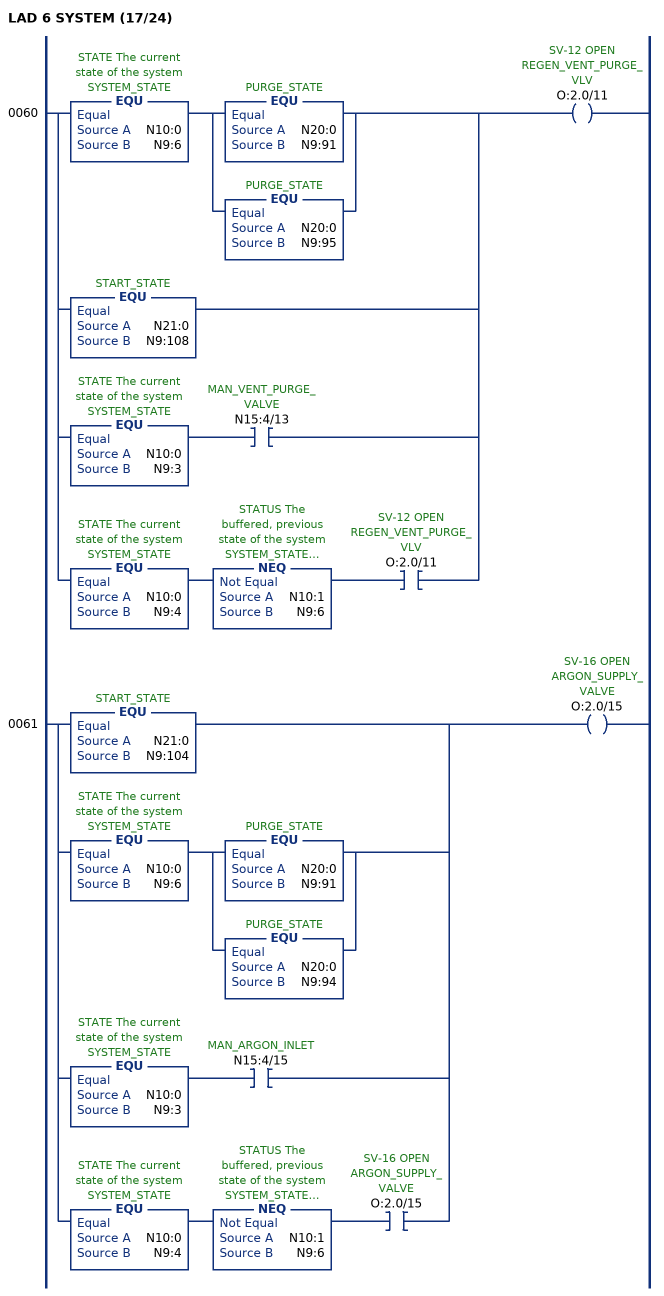
% Rung: 60 %
SOR BST EQU N10:0 N9:6 BST EQU N20:0 N9:91 NXB EQU N20:0 N9:95 BND NXB EQU N21:0 N9:108 NXB EQU N10:0 N9:3 XIC N15:4/13 NXB EQU N10:0 N9:4 NEQ N10:1 N9:6 XIC O:2.0/11 BND OTE O:2.0/11 EOR
%   N10:0  SYSTEM_STATE  "STATE The current state of the system" %
%   N9:6  SYSTEM_PURGE %
%   N20:0  PURGE_STATE %
%   N9:91  PURGE_INIT_VENT %
%   N9:95  PURGE_FINAL_VENT %
%   N21:0  START_STATE %
%   N9:108  START_VENT_GET_2 %
%   N9:3  SYSTEM_MANUAL  "STATE System Manual" %
%   N15:4/13  MAN_VENT_PURGE_VALVE %
%   N9:4  SYSTEM_ALARM  "STATE System Alarm" %
%   N10:1  SYSTEM_STATE_BUFFER  "STATUS The buffered, previous state of the system" %
%   O:2.0/11  REGEN_VENT_PURGE_VLV  "SV-12 OPEN" %
% Rung: 61 %
SOR BST EQU N21:0 N9:104 NXB EQU N10:0 N9:6 BST EQU N20:0 N9:91 NXB EQU N20:0 N9:94 BND NXB EQU N10:0 N9:3 XIC N15:4/15 NXB EQU N10:0 N9:4 NEQ N10:1 N9:6 XIC O:2.0/15 BND OTE O:2.0/15 EOR
%   N21:0  START_STATE %
%   N9:104  START_HEAT %
%   N10:0  SYSTEM_STATE  "STATE The current state of the system" %
%   N9:6  SYSTEM_PURGE %
%   N20:0  PURGE_STATE %
%   N9:91  PURGE_INIT_VENT %
%   N9:94  PURGE_BACKFILL %
%   N9:3  SYSTEM_MANUAL  "STATE System Manual" %
%   N15:4/15  MAN_ARGON_INLET %
%   N9:4  SYSTEM_ALARM  "STATE System Alarm" %
%   N10:1  SYSTEM_STATE_BUFFER  "STATUS The buffered, previous state of the system" %
%   O:2.0/15  ARGON_SUPPLY_VALVE  "SV-16 OPEN" %

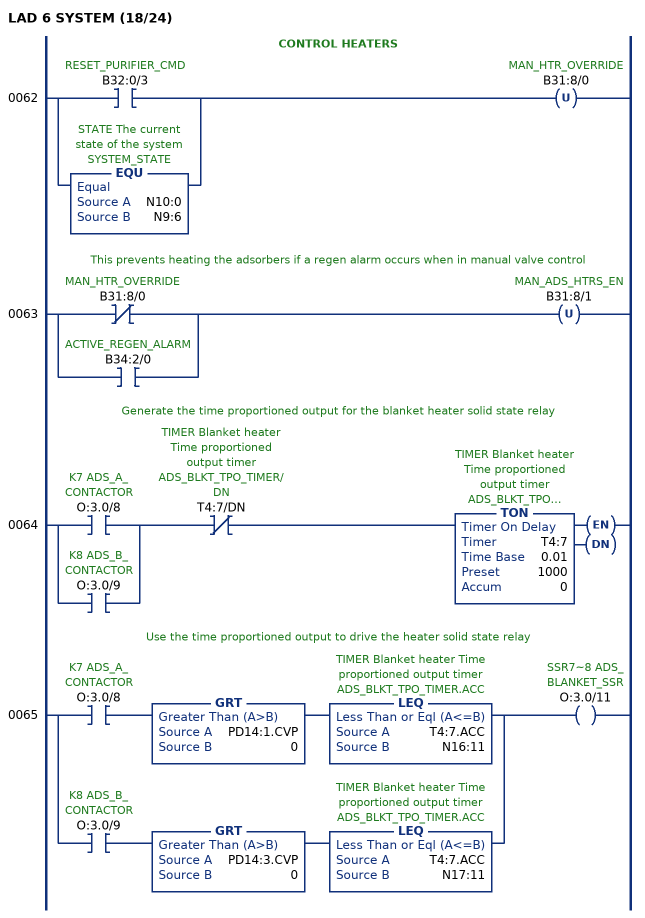
% Rung: 62 %
% TITLE: CONTROL HEATERS %
SOR BST XIC B32:0/3 NXB EQU N10:0 N9:6 BND OTU B31:8/0 EOR
%   B32:0/3  RESET_PURIFIER_CMD %
%   N10:0  SYSTEM_STATE  "STATE The current state of the system" %
%   N9:6  SYSTEM_PURGE %
%   B31:8/0  MAN_HTR_OVERRIDE %
% Rung: 63 %
% This prevents heating the adsorbers if a regen alarm occurs when in manual valve control %
SOR BST XIO B31:8/0 NXB XIC B34:2/0 BND OTU B31:8/1 EOR
%   B31:8/0  MAN_HTR_OVERRIDE %
%   B34:2/0  ACTIVE_REGEN_ALARM %
%   B31:8/1  MAN_ADS_HTRS_EN %
% Rung: 64 %
% Generate the time proportioned output for the blanket heater solid state relay %
SOR BST XIC O:3.0/8 NXB XIC O:3.0/9 BND XIO T4:7/DN TON T4:7 0.01 1000 0 EOR
%   O:3.0/8  ADS_A_CONTACTOR  "K7" %
%   O:3.0/9  ADS_B_CONTACTOR  "K8" %
%   T4:7  ADS_BLKT_TPO_TIMER  "TIMER Blanket heater Time proportioned output timer" %
% Rung: 65 %
% Use the time proportioned output to drive the heater solid state relay %
SOR BST XIC O:3.0/8 GRT PD14:1.CVP 0 LEQ T4:7.ACC N16:11 NXB XIC O:3.0/9 GRT PD14:3.CVP 0 LEQ T4:7.ACC N17:11 BND OTE O:3.0/11 EOR
%   O:3.0/8  ADS_A_CONTACTOR  "K7" %
%   T4:7  ADS_BLKT_TPO_TIMER  "TIMER Blanket heater Time proportioned output timer" %
%   N16:11  ADS_A_BLNKT_OUTPUT  "<datalog> CONTROL ADS A Blanket output (percent)" %
%   O:3.0/9  ADS_B_CONTACTOR  "K8" %
%   N17:11  ADS_B_BLNKT_OUTPUT  "<datalog> CONTROL ADS A Blanket output" %
%   O:3.0/11  ADS_BLANKET_SSR  "SSR7~8" %

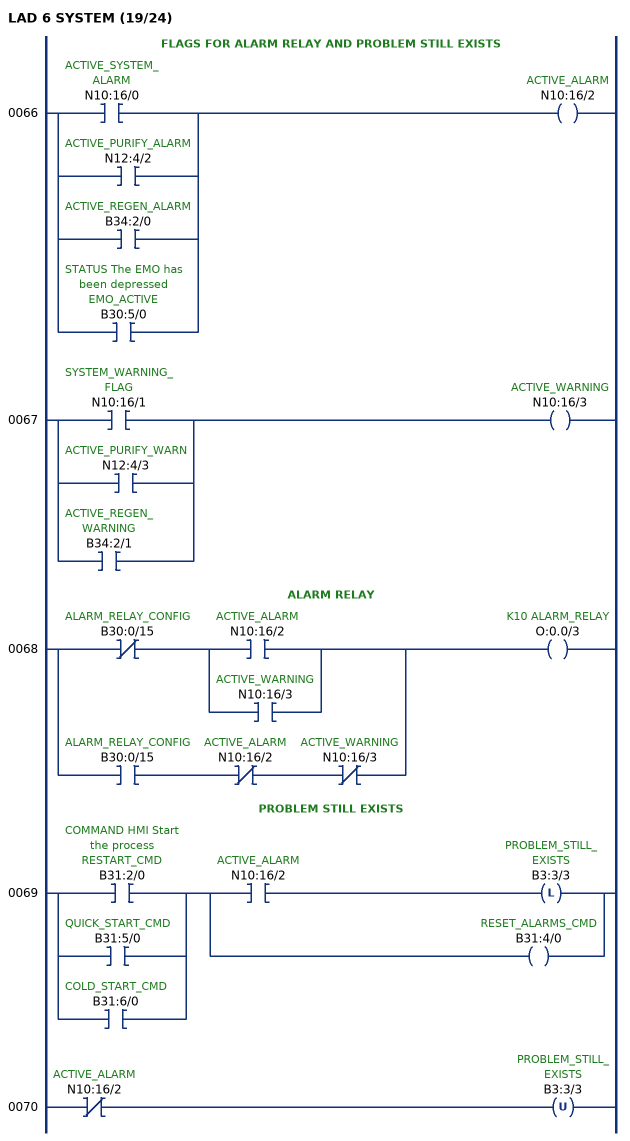
% Rung: 66 %
% TITLE: FLAGS FOR ALARM RELAY AND PROBLEM STILL EXISTS %
SOR BST XIC N10:16/0 NXB XIC N12:4/2 NXB XIC B34:2/0 NXB XIC B30:5/0 BND OTE N10:16/2 EOR
%   N10:16/0  ACTIVE_SYSTEM_ALARM %
%   N12:4/2  ACTIVE_PURIFY_ALARM %
%   B34:2/0  ACTIVE_REGEN_ALARM %
%   B30:5/0  EMO_ACTIVE  "STATUS The EMO has been depressed" %
%   N10:16/2  ACTIVE_ALARM %
% Rung: 67 %
SOR BST XIC N10:16/1 NXB XIC N12:4/3 NXB XIC B34:2/1 BND OTE N10:16/3 EOR
%   N10:16/1  SYSTEM_WARNING_FLAG %
%   N12:4/3  ACTIVE_PURIFY_WARN %
%   B34:2/1  ACTIVE_REGEN_WARNING %
%   N10:16/3  ACTIVE_WARNING %
% Rung: 68 %
% TITLE: ALARM RELAY %
SOR BST XIO B30:0/15 BST XIC N10:16/2 NXB XIC N10:16/3 BND NXB XIC B30:0/15 XIO N10:16/2 XIO N10:16/3 BND OTE O:0.0/3 EOR
%   B30:0/15  ALARM_RELAY_CONFIG %
%   N10:16/2  ACTIVE_ALARM %
%   N10:16/3  ACTIVE_WARNING %
%   O:0.0/3  ALARM_RELAY  "K10" %
% Rung: 69 %
% TITLE: PROBLEM STILL EXISTS %
SOR BST XIC B31:2/0 NXB XIC B31:5/0 NXB XIC B31:6/0 BND BST XIC N10:16/2 OTL B3:3/3 NXB OTE B31:4/0 BND EOR
%   B31:2/0  RESTART_CMD  "COMMAND HMI Start the process" %
%   B31:5/0  QUICK_START_CMD %
%   B31:6/0  COLD_START_CMD %
%   N10:16/2  ACTIVE_ALARM %
%   B3:3/3  PROBLEM_STILL_EXISTS %
%   B31:4/0  RESET_ALARMS_CMD %
% Rung: 70 %
SOR XIO N10:16/2 OTU B3:3/3 EOR
%   N10:16/2  ACTIVE_ALARM %
%   B3:3/3  PROBLEM_STILL_EXISTS %

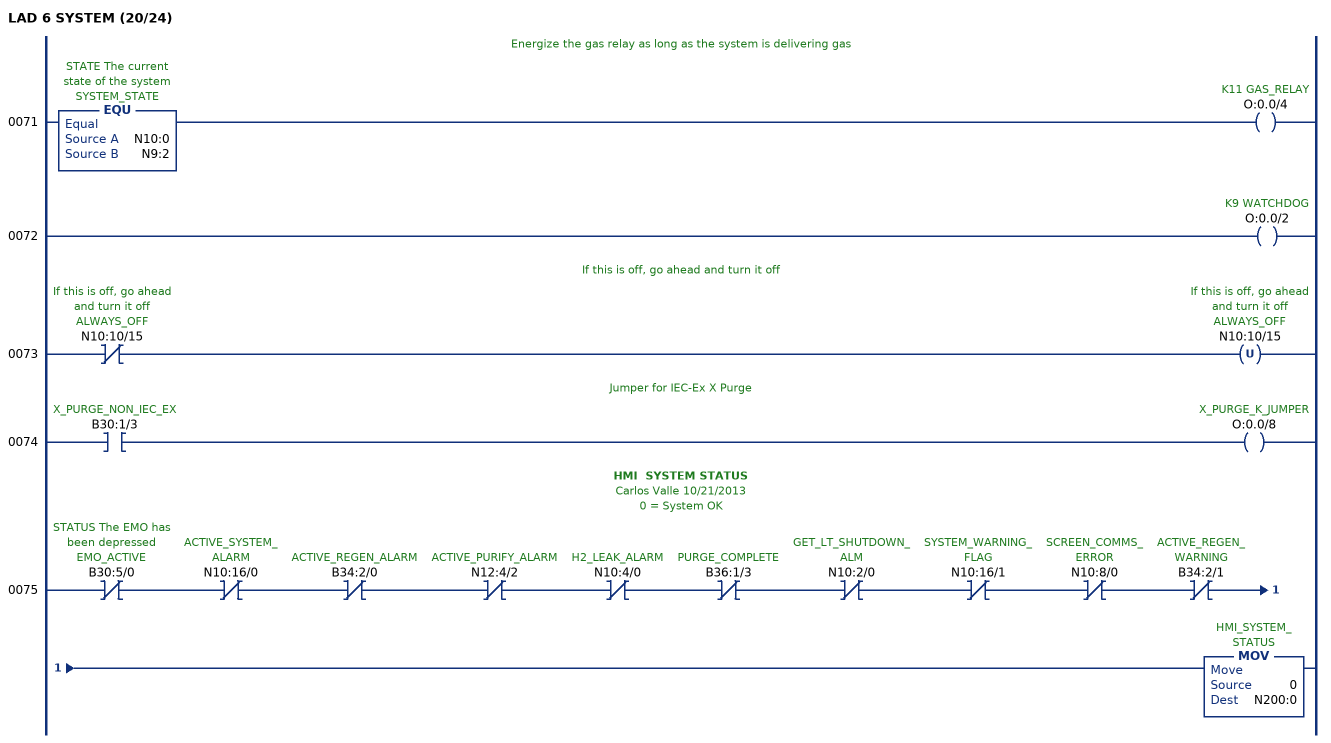
% Rung: 71 %
% Energize the gas relay as long as the system is delivering gas %
SOR EQU N10:0 N9:2 OTE O:0.0/4 EOR
%   N10:0  SYSTEM_STATE  "STATE The current state of the system" %
%   N9:2  SYSTEM_PROCESS  "STATE System Process" %
%   O:0.0/4  GAS_RELAY  "K11" %
% Rung: 72 %
SOR OTE O:0.0/2 EOR
%   O:0.0/2  WATCHDOG  "K9" %
% Rung: 73 %
% If this is off, go ahead and turn it off %
SOR XIO N10:10/15 OTU N10:10/15 EOR
%   N10:10/15  ALWAYS_OFF  "If this is off, go ahead and turn it off" %
% Rung: 74 %
% Jumper for IEC-Ex X Purge %
SOR XIC B30:1/3 OTE O:0.0/8 EOR
%   B30:1/3  X_PURGE_NON_IEC_EX %
%   O:0.0/8  X_PURGE_K_JUMPER %
% Rung: 75 %
% TITLE: HMI  SYSTEM STATUS %
% Carlos Valle 10/21/2013
% 0 = System OK %
SOR XIO B30:5/0 XIO N10:16/0 XIO B34:2/0 XIO N12:4/2 XIO N10:4/0 XIO B36:1/3 XIO N10:2/0 XIO N10:16/1 XIO N10:8/0 XIO B34:2/1 MOV 0 N200:0 EOR
%   B30:5/0  EMO_ACTIVE  "STATUS The EMO has been depressed" %
%   N10:16/0  ACTIVE_SYSTEM_ALARM %
%   B34:2/0  ACTIVE_REGEN_ALARM %
%   N12:4/2  ACTIVE_PURIFY_ALARM %
%   N10:4/0  H2_LEAK_ALARM %
%   B36:1/3  PURGE_COMPLETE %
%   N10:2/0  GET_LT_SHUTDOWN_ALM %
%   N10:16/1  SYSTEM_WARNING_FLAG %
%   N10:8/0  SCREEN_COMMS_ERROR %
%   B34:2/1  ACTIVE_REGEN_WARNING %
%   N200:0  HMI_SYSTEM_STATUS %

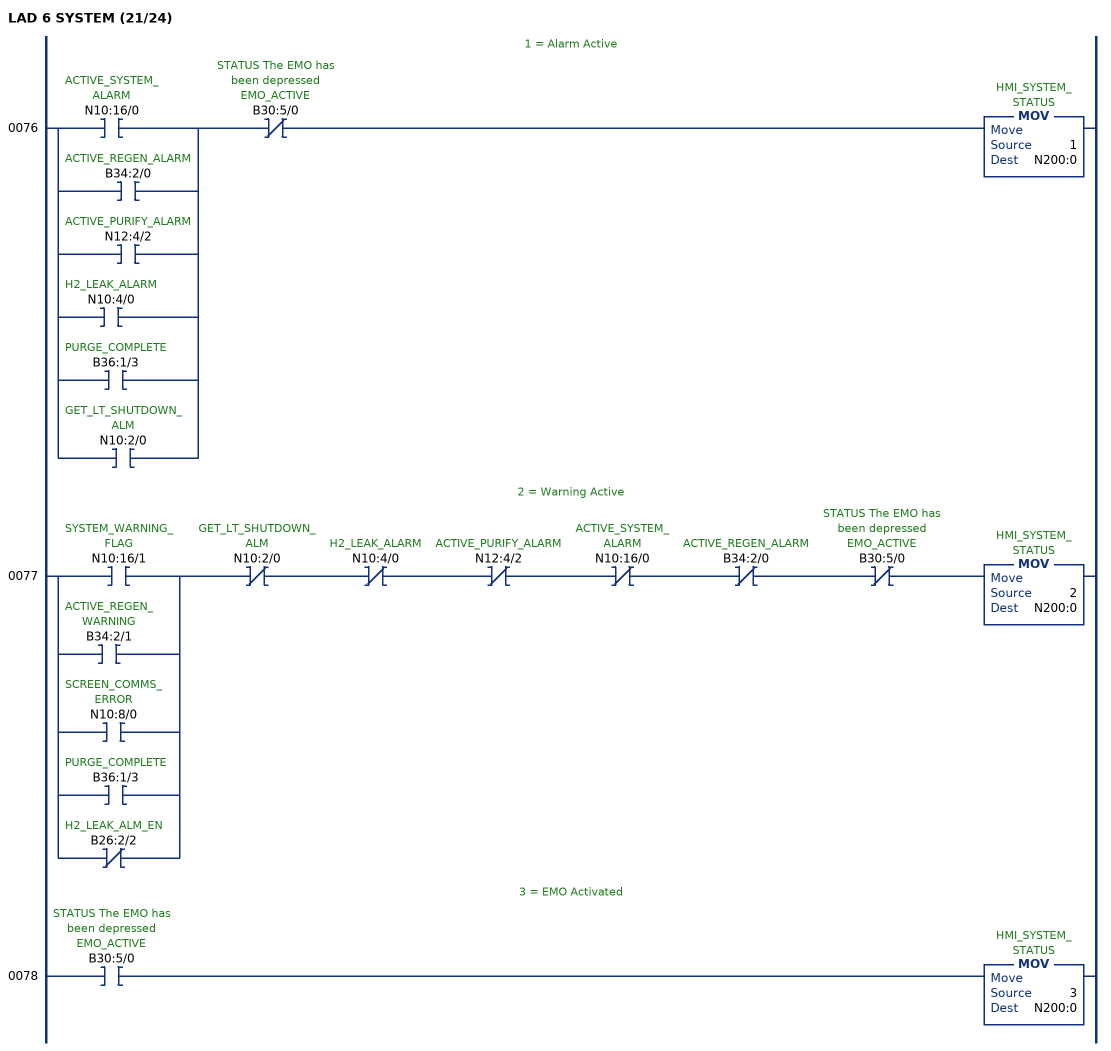
% Rung: 76 %
% 1 = Alarm Active %
SOR BST XIC N10:16/0 NXB XIC B34:2/0 NXB XIC N12:4/2 NXB XIC N10:4/0 NXB XIC B36:1/3 NXB XIC N10:2/0 BND XIO B30:5/0 MOV 1 N200:0 EOR
%   N10:16/0  ACTIVE_SYSTEM_ALARM %
%   B34:2/0  ACTIVE_REGEN_ALARM %
%   N12:4/2  ACTIVE_PURIFY_ALARM %
%   N10:4/0  H2_LEAK_ALARM %
%   B36:1/3  PURGE_COMPLETE %
%   N10:2/0  GET_LT_SHUTDOWN_ALM %
%   B30:5/0  EMO_ACTIVE  "STATUS The EMO has been depressed" %
%   N200:0  HMI_SYSTEM_STATUS %
% Rung: 77 %
% 2 = Warning Active %
SOR BST XIC N10:16/1 NXB XIC B34:2/1 NXB XIC N10:8/0 NXB XIC B36:1/3 NXB XIO B26:2/2 BND XIO N10:2/0 XIO N10:4/0 XIO N12:4/2 XIO N10:16/0 XIO B34:2/0 XIO B30:5/0 MOV 2 N200:0 EOR
%   N10:16/1  SYSTEM_WARNING_FLAG %
%   B34:2/1  ACTIVE_REGEN_WARNING %
%   N10:8/0  SCREEN_COMMS_ERROR %
%   B36:1/3  PURGE_COMPLETE %
%   B26:2/2  H2_LEAK_ALM_EN %
%   N10:2/0  GET_LT_SHUTDOWN_ALM %
%   N10:4/0  H2_LEAK_ALARM %
%   N12:4/2  ACTIVE_PURIFY_ALARM %
%   N10:16/0  ACTIVE_SYSTEM_ALARM %
%   B34:2/0  ACTIVE_REGEN_ALARM %
%   B30:5/0  EMO_ACTIVE  "STATUS The EMO has been depressed" %
%   N200:0  HMI_SYSTEM_STATUS %
% Rung: 78 %
% 3 = EMO Activated %
SOR XIC B30:5/0 MOV 3 N200:0 EOR
%   B30:5/0  EMO_ACTIVE  "STATUS The EMO has been depressed" %
%   N200:0  HMI_SYSTEM_STATUS %

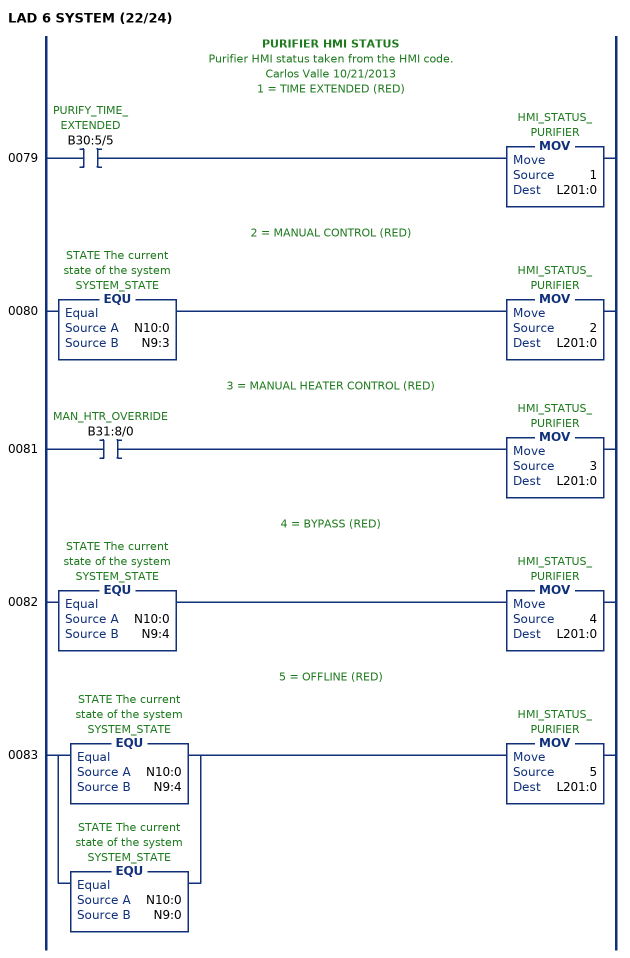
% Rung: 79 %
% TITLE: PURIFIER HMI STATUS %
% Purifier HMI status taken from the HMI code.
% Carlos Valle 10/21/2013
% 1 = TIME EXTENDED (RED) %
SOR XIC B30:5/5 MOV 1 L201:0 EOR
%   B30:5/5  PURIFY_TIME_EXTENDED %
%   L201:0  HMI_STATUS_PURIFIER %
% Rung: 80 %
% 2 = MANUAL CONTROL (RED) %
SOR EQU N10:0 N9:3 MOV 2 L201:0 EOR
%   N10:0  SYSTEM_STATE  "STATE The current state of the system" %
%   N9:3  SYSTEM_MANUAL  "STATE System Manual" %
%   L201:0  HMI_STATUS_PURIFIER %
% Rung: 81 %
% 3 = MANUAL HEATER CONTROL (RED) %
SOR XIC B31:8/0 MOV 3 L201:0 EOR
%   B31:8/0  MAN_HTR_OVERRIDE %
%   L201:0  HMI_STATUS_PURIFIER %
% Rung: 82 %
% 4 = BYPASS (RED) %
SOR EQU N10:0 N9:4 MOV 4 L201:0 EOR
%   N10:0  SYSTEM_STATE  "STATE The current state of the system" %
%   N9:4  SYSTEM_ALARM  "STATE System Alarm" %
%   L201:0  HMI_STATUS_PURIFIER %
% Rung: 83 %
% 5 = OFFLINE (RED) %
SOR BST EQU N10:0 N9:4 NXB EQU N10:0 N9:0 BND MOV 5 L201:0 EOR
%   N10:0  SYSTEM_STATE  "STATE The current state of the system" %
%   N9:4  SYSTEM_ALARM  "STATE System Alarm" %
%   N9:0  SYSTEM_OFFLINE %
%   L201:0  HMI_STATUS_PURIFIER %

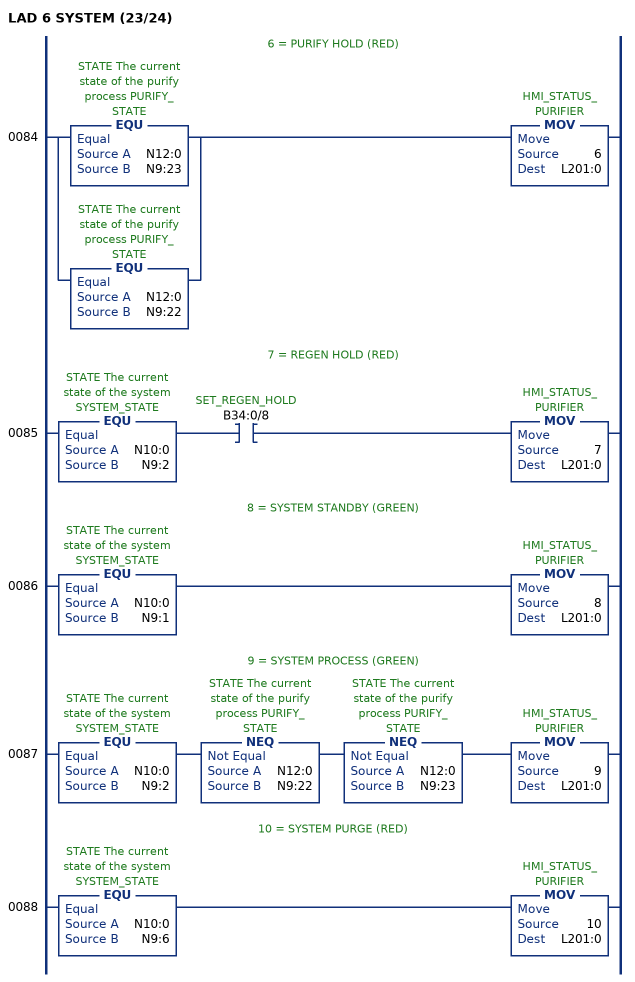
% Rung: 84 %
% 6 = PURIFY HOLD (RED) %
SOR BST EQU N12:0 N9:23 NXB EQU N12:0 N9:22 BND MOV 6 L201:0 EOR
%   N12:0  PURIFY_STATE  "STATE The current state of the purify process" %
%   N9:23  PURIFY_MANUAL_HOLD  "STATE Purify Manual Hold" %
%   N9:22  PURIFY_HOLD  "STATE Purify Hold" %
%   L201:0  HMI_STATUS_PURIFIER %
% Rung: 85 %
% 7 = REGEN HOLD (RED) %
SOR EQU N10:0 N9:2 XIC B34:0/8 MOV 7 L201:0 EOR
%   N10:0  SYSTEM_STATE  "STATE The current state of the system" %
%   N9:2  SYSTEM_PROCESS  "STATE System Process" %
%   B34:0/8  SET_REGEN_HOLD %
%   L201:0  HMI_STATUS_PURIFIER %
% Rung: 86 %
% 8 = SYSTEM STANDBY (GREEN) %
SOR EQU N10:0 N9:1 MOV 8 L201:0 EOR
%   N10:0  SYSTEM_STATE  "STATE The current state of the system" %
%   N9:1  SYSTEM_STANDBY  "STATE System Process" %
%   L201:0  HMI_STATUS_PURIFIER %
% Rung: 87 %
% 9 = SYSTEM PROCESS (GREEN) %
SOR EQU N10:0 N9:2 NEQ N12:0 N9:22 NEQ N12:0 N9:23 MOV 9 L201:0 EOR
%   N10:0  SYSTEM_STATE  "STATE The current state of the system" %
%   N9:2  SYSTEM_PROCESS  "STATE System Process" %
%   N12:0  PURIFY_STATE  "STATE The current state of the purify process" %
%   N9:22  PURIFY_HOLD  "STATE Purify Hold" %
%   N9:23  PURIFY_MANUAL_HOLD  "STATE Purify Manual Hold" %
%   L201:0  HMI_STATUS_PURIFIER %
% Rung: 88 %
% 10 = SYSTEM PURGE (RED) %
SOR EQU N10:0 N9:6 MOV 10 L201:0 EOR
%   N10:0  SYSTEM_STATE  "STATE The current state of the system" %
%   N9:6  SYSTEM_PURGE %
%   L201:0  HMI_STATUS_PURIFIER %

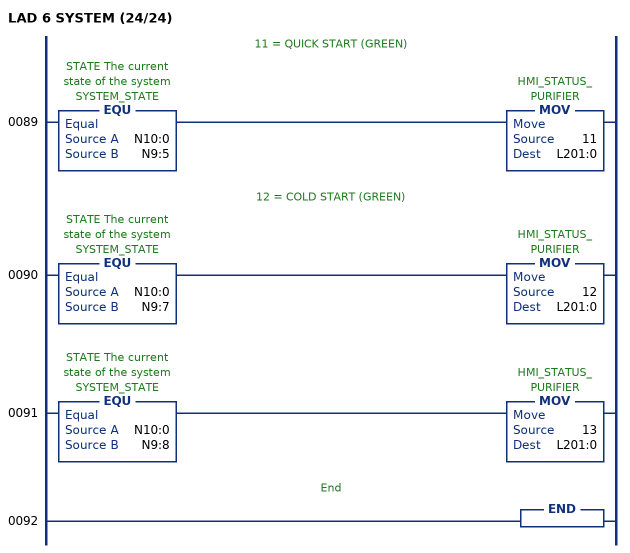
% Rung: 89 %
% 11 = QUICK START (GREEN) %
SOR EQU N10:0 N9:5 MOV 11 L201:0 EOR
%   N10:0  SYSTEM_STATE  "STATE The current state of the system" %
%   N9:5  SYSTEM_QUICK_START %
%   L201:0  HMI_STATUS_PURIFIER %
% Rung: 90 %
% 12 = COLD START (GREEN) %
SOR EQU N10:0 N9:7 MOV 12 L201:0 EOR
%   N10:0  SYSTEM_STATE  "STATE The current state of the system" %
%   N9:7  SYSTEM_COLD_START %
%   L201:0  HMI_STATUS_PURIFIER %
% Rung: 91 %
SOR EQU N10:0 N9:8 MOV 13 L201:0 EOR
%   N10:0  SYSTEM_STATE  "STATE The current state of the system" %
%   N9:8  SYSTEM_SUPPLEMENTAL %
%   L201:0  HMI_STATUS_PURIFIER %
% Rung: 92 %
% End %
SOR END EOR

LADDER 7 "PROCESSING"    % Runs the processing control %
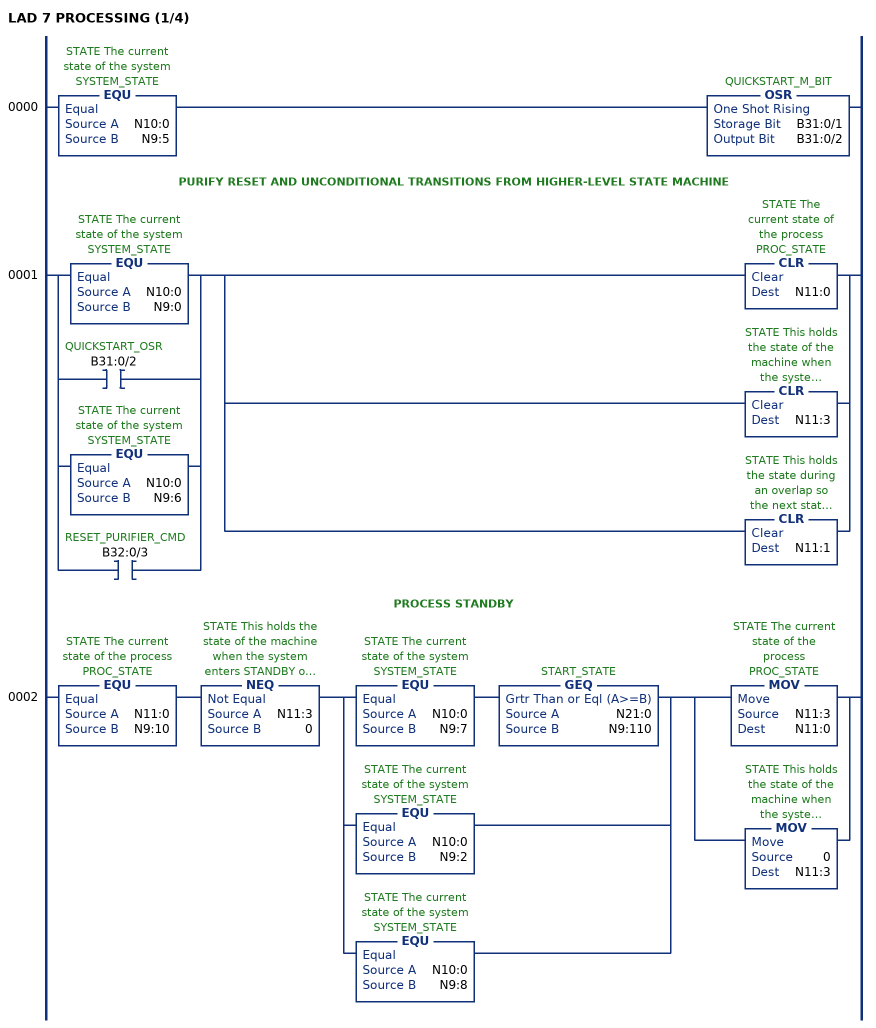
% Rung: 0 %
SOR EQU N10:0 N9:5 OSR B31:0/1 B31:0/2 EOR
%   N10:0  SYSTEM_STATE  "STATE The current state of the system" %
%   N9:5  SYSTEM_QUICK_START %
%   B31:0/1  QUICKSTART_M_BIT %
%   B31:0/2  QUICKSTART_OSR %
% Rung: 1 %
% TITLE: PURIFY RESET AND UNCONDITIONAL TRANSITIONS FROM HIGHER-LEVEL STATE MACHINE %
SOR BST EQU N10:0 N9:0 NXB XIC B31:0/2 NXB EQU N10:0 N9:6 NXB XIC B32:0/3 BND BST CLR N11:0 NXB CLR N11:3 NXB CLR N11:1 BND EOR
%   N10:0  SYSTEM_STATE  "STATE The current state of the system" %
%   N9:0  SYSTEM_OFFLINE %
%   B31:0/2  QUICKSTART_OSR %
%   N9:6  SYSTEM_PURGE %
%   B32:0/3  RESET_PURIFIER_CMD %
%   N11:0  PROC_STATE  "STATE The current state of the process" %
%   N11:3  PROC_STATE_BUFFER  "STATE This holds the state of the machine when the system enters STANDBY or ALARM" %
%   N11:1  PROC_OVERLAP_BUFFER  "STATE This holds the state during an overlap so the next state can be determined" %
% Rung: 2 %
% TITLE: PROCESS STANDBY %
SOR EQU N11:0 N9:10 NEQ N11:3 0 BST EQU N10:0 N9:7 GEQ N21:0 N9:110 NXB EQU N10:0 N9:2 NXB EQU N10:0 N9:8 BND BST MOV N11:3 N11:0 NXB MOV 0 N11:3 BND EOR
%   N11:0  PROC_STATE  "STATE The current state of the process" %
%   N9:10  PROC_STANDBY  "STATE Process Standby" %
%   N11:3  PROC_STATE_BUFFER  "STATE This holds the state of the machine when the system enters STANDBY or ALARM" %
%   N10:0  SYSTEM_STATE  "STATE The current state of the system" %
%   N9:7  SYSTEM_COLD_START %
%   N21:0  START_STATE %
%   N9:110  START_REG_VENT %
%   N9:2  SYSTEM_PROCESS  "STATE System Process" %
%   N9:8  SYSTEM_SUPPLEMENTAL %

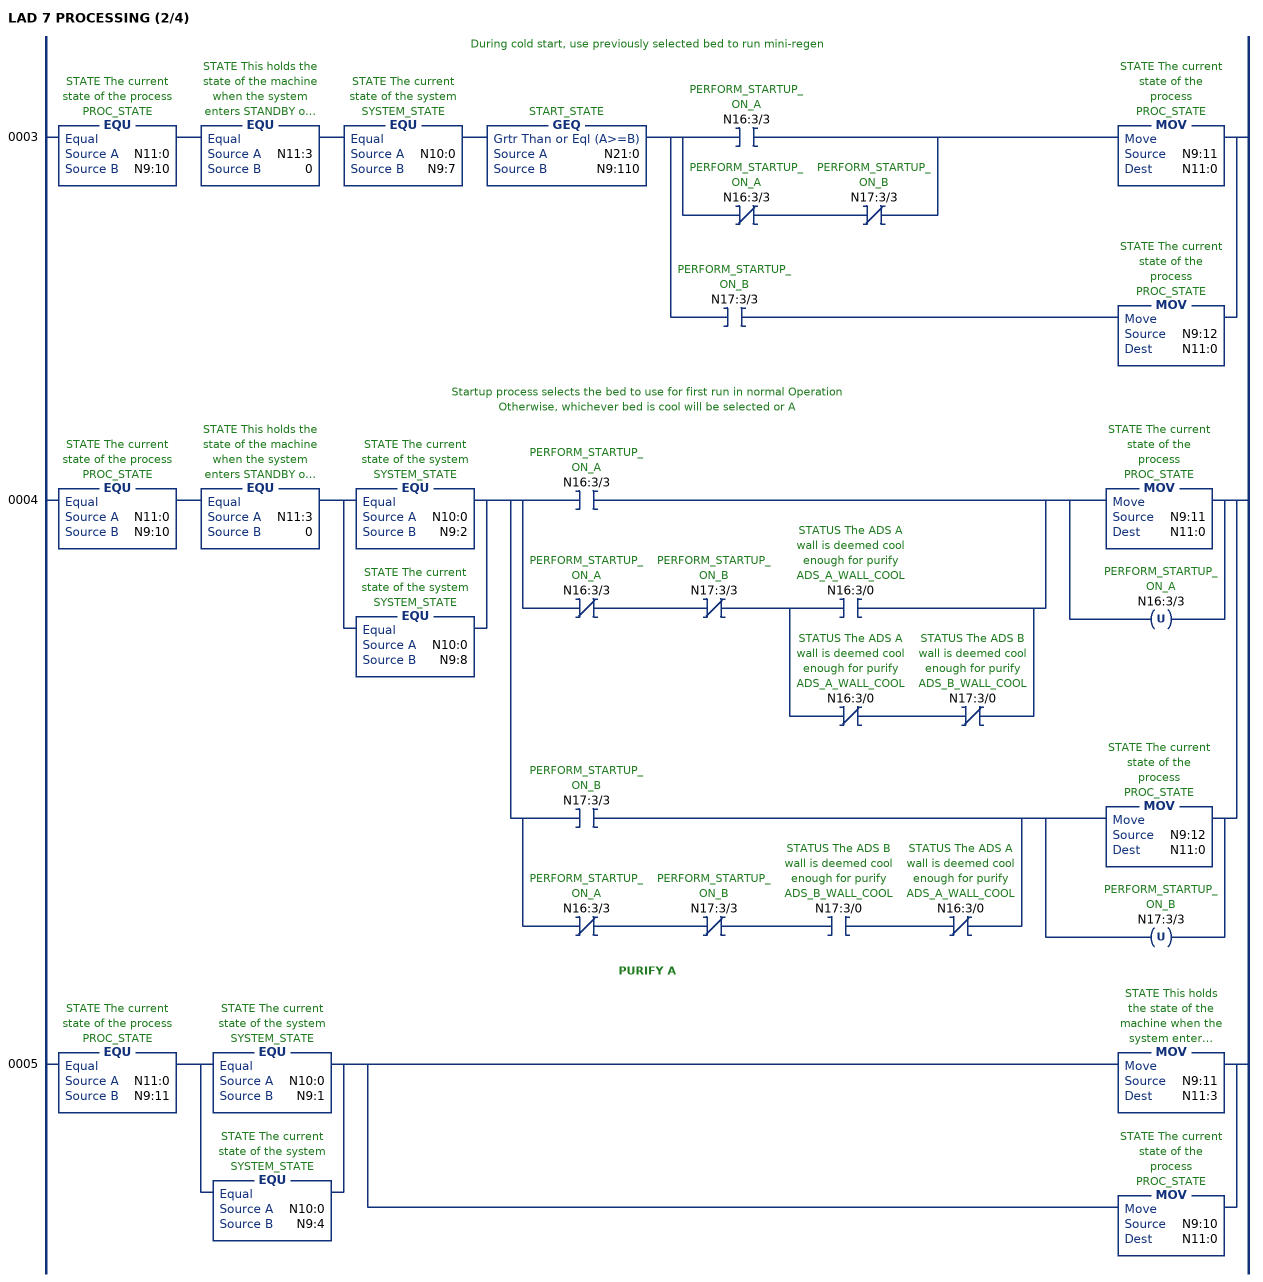
% Rung: 3 %
% During cold start, use previously selected bed to run mini-regen %
SOR EQU N11:0 N9:10 EQU N11:3 0 EQU N10:0 N9:7 GEQ N21:0 N9:110 BST BST XIC N16:3/3 NXB XIO N16:3/3 XIO N17:3/3 BND MOV N9:11 N11:0 NXB XIC N17:3/3 MOV N9:12 N11:0 BND EOR
%   N11:0  PROC_STATE  "STATE The current state of the process" %
%   N9:10  PROC_STANDBY  "STATE Process Standby" %
%   N11:3  PROC_STATE_BUFFER  "STATE This holds the state of the machine when the system enters STANDBY or ALARM" %
%   N10:0  SYSTEM_STATE  "STATE The current state of the system" %
%   N9:7  SYSTEM_COLD_START %
%   N21:0  START_STATE %
%   N9:110  START_REG_VENT %
%   N16:3/3  PERFORM_STARTUP_ON_A %
%   N17:3/3  PERFORM_STARTUP_ON_B %
%   N9:11  PROC_PFY_A_REG_B  "STATE Process Purify A" %
%   N9:12  PROC_PFY_B_REG_A  "STATE Process Purify B" %
% Rung: 4 %
% Startup process selects the bed to use for first run in normal Operation
% Otherwise, whichever bed is cool will be selected or A %
SOR EQU N11:0 N9:10 EQU N11:3 0 BST EQU N10:0 N9:2 NXB EQU N10:0 N9:8 BND BST BST XIC N16:3/3 NXB XIO N16:3/3 XIO N17:3/3 BST XIC N16:3/0 NXB XIO N16:3/0 XIO N17:3/0 BND BND BST MOV N9:11 N11:0 NXB OTU N16:3/3 BND NXB BST XIC N17:3/3 NXB XIO N16:3/3 XIO N17:3/3 XIC N17:3/0 XIO N16:3/0 BND BST MOV N9:12 N11:0 NXB OTU N17:3/3 BND BND EOR
%   N11:0  PROC_STATE  "STATE The current state of the process" %
%   N9:10  PROC_STANDBY  "STATE Process Standby" %
%   N11:3  PROC_STATE_BUFFER  "STATE This holds the state of the machine when the system enters STANDBY or ALARM" %
%   N10:0  SYSTEM_STATE  "STATE The current state of the system" %
%   N9:2  SYSTEM_PROCESS  "STATE System Process" %
%   N9:8  SYSTEM_SUPPLEMENTAL %
%   N16:3/3  PERFORM_STARTUP_ON_A %
%   N17:3/3  PERFORM_STARTUP_ON_B %
%   N16:3/0  ADS_A_WALL_COOL  "STATUS The ADS A wall is deemed cool enough for purify" %
%   N17:3/0  ADS_B_WALL_COOL  "STATUS The ADS B wall is deemed cool enough for purify" %
%   N9:11  PROC_PFY_A_REG_B  "STATE Process Purify A" %
%   N9:12  PROC_PFY_B_REG_A  "STATE Process Purify B" %
% Rung: 5 %
% TITLE: PURIFY A %
SOR EQU N11:0 N9:11 BST EQU N10:0 N9:1 NXB EQU N10:0 N9:4 BND BST MOV N9:11 N11:3 NXB MOV N9:10 N11:0 BND EOR
%   N11:0  PROC_STATE  "STATE The current state of the process" %
%   N9:11  PROC_PFY_A_REG_B  "STATE Process Purify A" %
%   N10:0  SYSTEM_STATE  "STATE The current state of the system" %
%   N9:1  SYSTEM_STANDBY  "STATE System Process" %
%   N9:4  SYSTEM_ALARM  "STATE System Alarm" %
%   N11:3  PROC_STATE_BUFFER  "STATE This holds the state of the machine when the system enters STANDBY or ALARM" %
%   N9:10  PROC_STANDBY  "STATE Process Standby" %

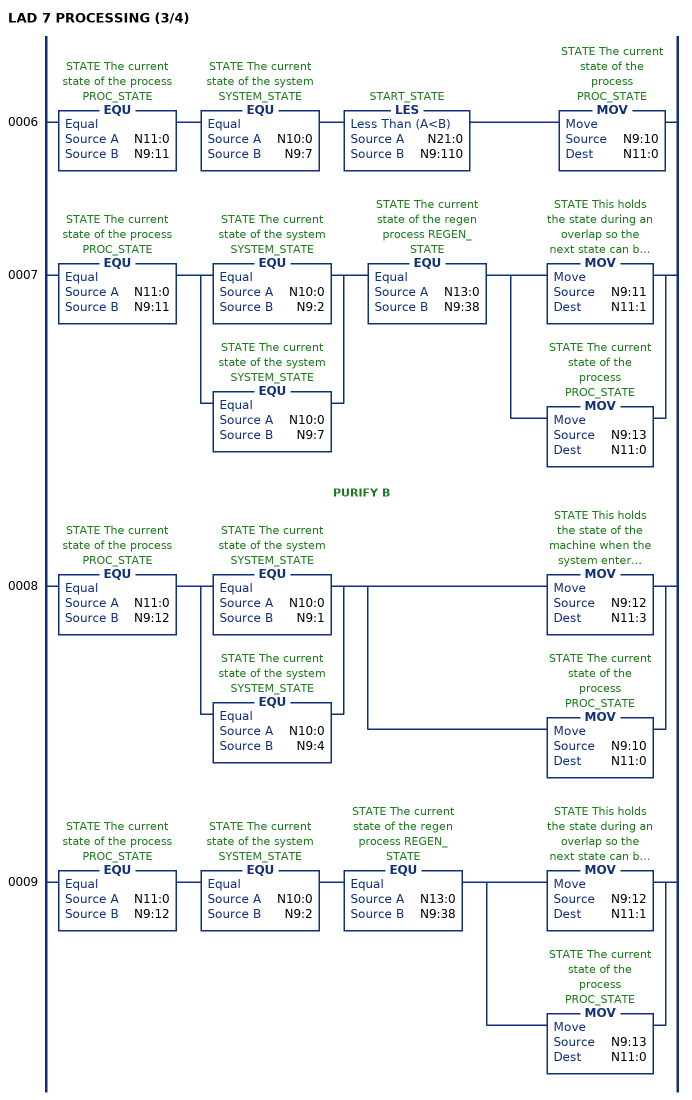
% Rung: 6 %
SOR EQU N11:0 N9:11 EQU N10:0 N9:7 LES N21:0 N9:110 MOV N9:10 N11:0 EOR
%   N11:0  PROC_STATE  "STATE The current state of the process" %
%   N9:11  PROC_PFY_A_REG_B  "STATE Process Purify A" %
%   N10:0  SYSTEM_STATE  "STATE The current state of the system" %
%   N9:7  SYSTEM_COLD_START %
%   N21:0  START_STATE %
%   N9:110  START_REG_VENT %
%   N9:10  PROC_STANDBY  "STATE Process Standby" %
% Rung: 7 %
SOR EQU N11:0 N9:11 BST EQU N10:0 N9:2 NXB EQU N10:0 N9:7 BND EQU N13:0 N9:38 BST MOV N9:11 N11:1 NXB MOV N9:13 N11:0 BND EOR
%   N11:0  PROC_STATE  "STATE The current state of the process" %
%   N9:11  PROC_PFY_A_REG_B  "STATE Process Purify A" %
%   N10:0  SYSTEM_STATE  "STATE The current state of the system" %
%   N9:2  SYSTEM_PROCESS  "STATE System Process" %
%   N9:7  SYSTEM_COLD_START %
%   N13:0  REGEN_STATE  "STATE The current state of the regen process" %
%   N9:38  REGEN_DONE %
%   N11:1  PROC_OVERLAP_BUFFER  "STATE This holds the state during an overlap so the next state can be determined" %
%   N9:13  PROC_OVERLAP  "STATE Process Purify Overlap" %
% Rung: 8 %
% TITLE: PURIFY B %
SOR EQU N11:0 N9:12 BST EQU N10:0 N9:1 NXB EQU N10:0 N9:4 BND BST MOV N9:12 N11:3 NXB MOV N9:10 N11:0 BND EOR
%   N11:0  PROC_STATE  "STATE The current state of the process" %
%   N9:12  PROC_PFY_B_REG_A  "STATE Process Purify B" %
%   N10:0  SYSTEM_STATE  "STATE The current state of the system" %
%   N9:1  SYSTEM_STANDBY  "STATE System Process" %
%   N9:4  SYSTEM_ALARM  "STATE System Alarm" %
%   N11:3  PROC_STATE_BUFFER  "STATE This holds the state of the machine when the system enters STANDBY or ALARM" %
%   N9:10  PROC_STANDBY  "STATE Process Standby" %
% Rung: 9 %
SOR EQU N11:0 N9:12 EQU N10:0 N9:2 EQU N13:0 N9:38 BST MOV N9:12 N11:1 NXB MOV N9:13 N11:0 BND EOR
%   N11:0  PROC_STATE  "STATE The current state of the process" %
%   N9:12  PROC_PFY_B_REG_A  "STATE Process Purify B" %
%   N10:0  SYSTEM_STATE  "STATE The current state of the system" %
%   N9:2  SYSTEM_PROCESS  "STATE System Process" %
%   N13:0  REGEN_STATE  "STATE The current state of the regen process" %
%   N9:38  REGEN_DONE %
%   N11:1  PROC_OVERLAP_BUFFER  "STATE This holds the state during an overlap so the next state can be determined" %
%   N9:13  PROC_OVERLAP  "STATE Process Purify Overlap" %

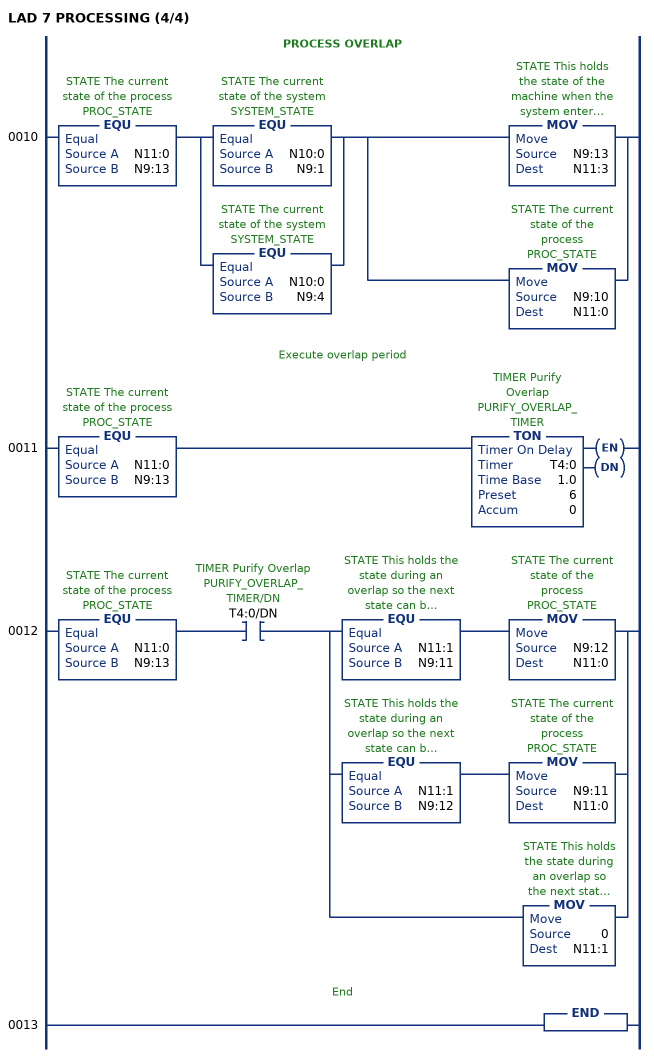
% Rung: 10 %
% TITLE: PROCESS OVERLAP %
SOR EQU N11:0 N9:13 BST EQU N10:0 N9:1 NXB EQU N10:0 N9:4 BND BST MOV N9:13 N11:3 NXB MOV N9:10 N11:0 BND EOR
%   N11:0  PROC_STATE  "STATE The current state of the process" %
%   N9:13  PROC_OVERLAP  "STATE Process Purify Overlap" %
%   N10:0  SYSTEM_STATE  "STATE The current state of the system" %
%   N9:1  SYSTEM_STANDBY  "STATE System Process" %
%   N9:4  SYSTEM_ALARM  "STATE System Alarm" %
%   N11:3  PROC_STATE_BUFFER  "STATE This holds the state of the machine when the system enters STANDBY or ALARM" %
%   N9:10  PROC_STANDBY  "STATE Process Standby" %
% Rung: 11 %
% Execute overlap period %
SOR EQU N11:0 N9:13 TON T4:0 1.0 6 0 EOR
%   N11:0  PROC_STATE  "STATE The current state of the process" %
%   N9:13  PROC_OVERLAP  "STATE Process Purify Overlap" %
%   T4:0  PURIFY_OVERLAP_TIMER  "TIMER Purify Overlap" %
% Rung: 12 %
SOR EQU N11:0 N9:13 XIC T4:0/DN BST EQU N11:1 N9:11 MOV N9:12 N11:0 NXB EQU N11:1 N9:12 MOV N9:11 N11:0 NXB MOV 0 N11:1 BND EOR
%   N11:0  PROC_STATE  "STATE The current state of the process" %
%   N9:13  PROC_OVERLAP  "STATE Process Purify Overlap" %
%   T4:0  PURIFY_OVERLAP_TIMER  "TIMER Purify Overlap" %
%   N11:1  PROC_OVERLAP_BUFFER  "STATE This holds the state during an overlap so the next state can be determined" %
%   N9:11  PROC_PFY_A_REG_B  "STATE Process Purify A" %
%   N9:12  PROC_PFY_B_REG_A  "STATE Process Purify B" %
% Rung: 13 %
% End %
SOR END EOR

LADDER 8 "MANUAL_CTL"    % Runs the manual valve control %
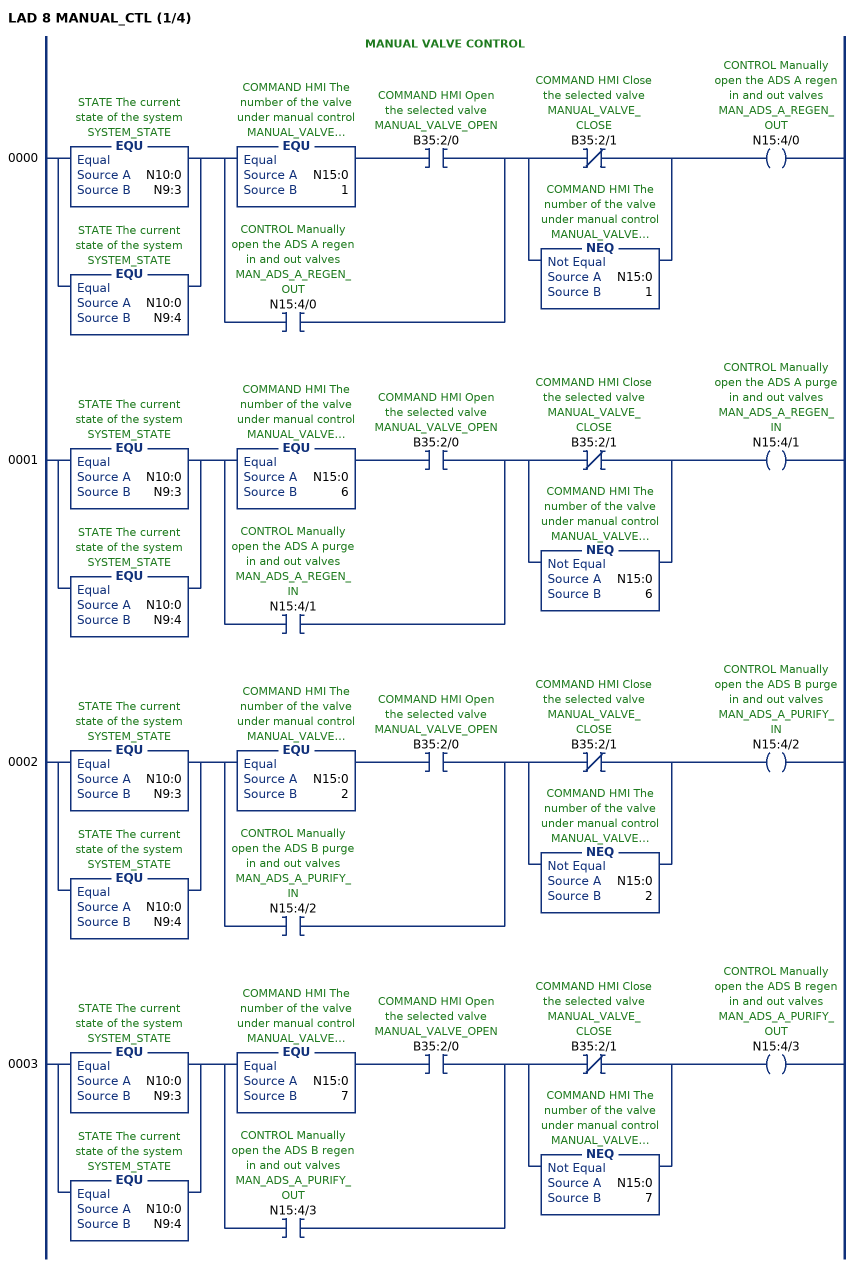
% Rung: 0 %
% TITLE: MANUAL VALVE CONTROL %
SOR BST EQU N10:0 N9:3 NXB EQU N10:0 N9:4 BND BST EQU N15:0 1 XIC B35:2/0 NXB XIC N15:4/0 BND BST XIO B35:2/1 NXB NEQ N15:0 1 BND OTE N15:4/0 EOR
%   N10:0  SYSTEM_STATE  "STATE The current state of the system" %
%   N9:3  SYSTEM_MANUAL  "STATE System Manual" %
%   N9:4  SYSTEM_ALARM  "STATE System Alarm" %
%   N15:0  MANUAL_VALVE_NUMBER  "COMMAND HMI The number of the valve under manual control" %
%   B35:2/0  MANUAL_VALVE_OPEN  "COMMAND HMI Open the selected valve" %
%   N15:4/0  MAN_ADS_A_REGEN_OUT  "CONTROL Manually open the ADS A regen in and out valves" %
%   B35:2/1  MANUAL_VALVE_CLOSE  "COMMAND HMI Close the selected valve" %
% Rung: 1 %
SOR BST EQU N10:0 N9:3 NXB EQU N10:0 N9:4 BND BST EQU N15:0 6 XIC B35:2/0 NXB XIC N15:4/1 BND BST XIO B35:2/1 NXB NEQ N15:0 6 BND OTE N15:4/1 EOR
%   N10:0  SYSTEM_STATE  "STATE The current state of the system" %
%   N9:3  SYSTEM_MANUAL  "STATE System Manual" %
%   N9:4  SYSTEM_ALARM  "STATE System Alarm" %
%   N15:0  MANUAL_VALVE_NUMBER  "COMMAND HMI The number of the valve under manual control" %
%   B35:2/0  MANUAL_VALVE_OPEN  "COMMAND HMI Open the selected valve" %
%   N15:4/1  MAN_ADS_A_REGEN_IN  "CONTROL Manually open the ADS A purge in and out valves" %
%   B35:2/1  MANUAL_VALVE_CLOSE  "COMMAND HMI Close the selected valve" %
% Rung: 2 %
SOR BST EQU N10:0 N9:3 NXB EQU N10:0 N9:4 BND BST EQU N15:0 2 XIC B35:2/0 NXB XIC N15:4/2 BND BST XIO B35:2/1 NXB NEQ N15:0 2 BND OTE N15:4/2 EOR
%   N10:0  SYSTEM_STATE  "STATE The current state of the system" %
%   N9:3  SYSTEM_MANUAL  "STATE System Manual" %
%   N9:4  SYSTEM_ALARM  "STATE System Alarm" %
%   N15:0  MANUAL_VALVE_NUMBER  "COMMAND HMI The number of the valve under manual control" %
%   B35:2/0  MANUAL_VALVE_OPEN  "COMMAND HMI Open the selected valve" %
%   N15:4/2  MAN_ADS_A_PURIFY_IN  "CONTROL Manually open the ADS B purge in and out valves" %
%   B35:2/1  MANUAL_VALVE_CLOSE  "COMMAND HMI Close the selected valve" %
% Rung: 3 %
SOR BST EQU N10:0 N9:3 NXB EQU N10:0 N9:4 BND BST EQU N15:0 7 XIC B35:2/0 NXB XIC N15:4/3 BND BST XIO B35:2/1 NXB NEQ N15:0 7 BND OTE N15:4/3 EOR
%   N10:0  SYSTEM_STATE  "STATE The current state of the system" %
%   N9:3  SYSTEM_MANUAL  "STATE System Manual" %
%   N9:4  SYSTEM_ALARM  "STATE System Alarm" %
%   N15:0  MANUAL_VALVE_NUMBER  "COMMAND HMI The number of the valve under manual control" %
%   B35:2/0  MANUAL_VALVE_OPEN  "COMMAND HMI Open the selected valve" %
%   N15:4/3  MAN_ADS_A_PURIFY_OUT  "CONTROL Manually open the ADS B regen in and out valves" %
%   B35:2/1  MANUAL_VALVE_CLOSE  "COMMAND HMI Close the selected valve" %

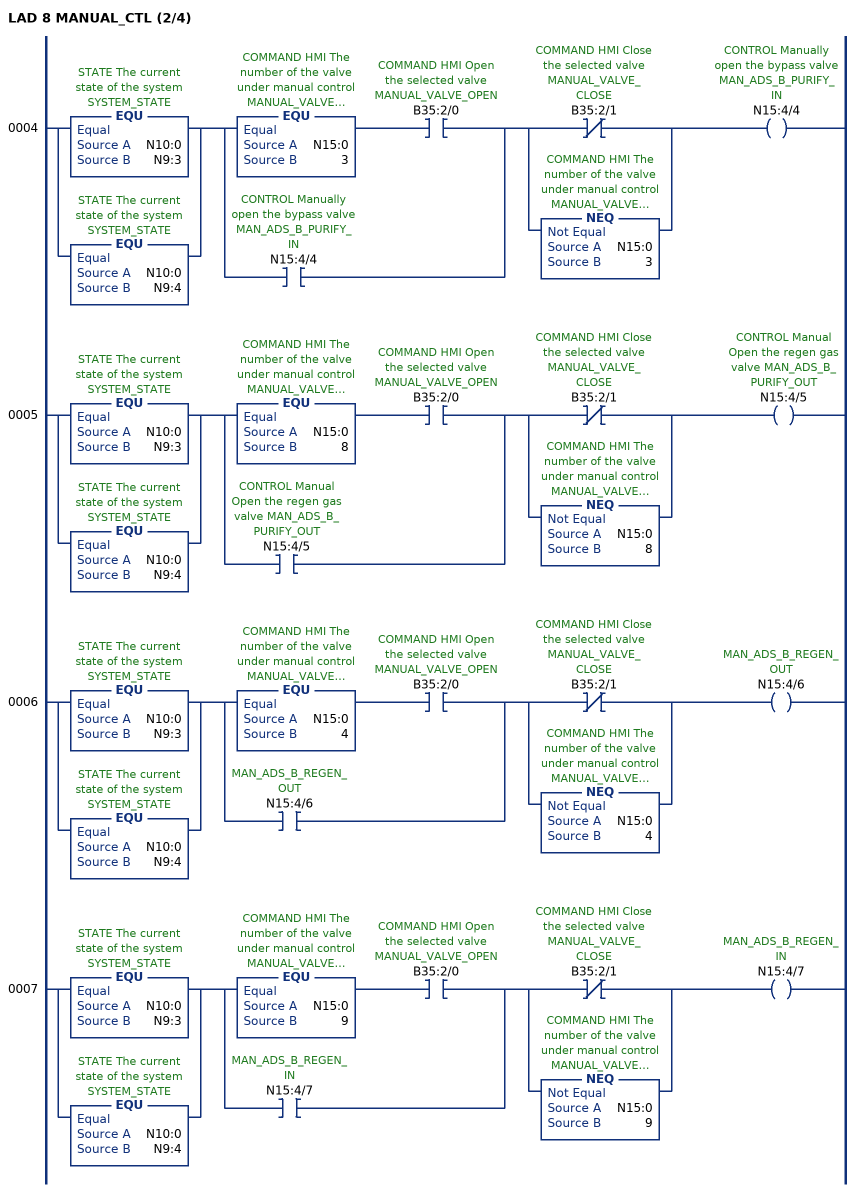
% Rung: 4 %
SOR BST EQU N10:0 N9:3 NXB EQU N10:0 N9:4 BND BST EQU N15:0 3 XIC B35:2/0 NXB XIC N15:4/4 BND BST XIO B35:2/1 NXB NEQ N15:0 3 BND OTE N15:4/4 EOR
%   N10:0  SYSTEM_STATE  "STATE The current state of the system" %
%   N9:3  SYSTEM_MANUAL  "STATE System Manual" %
%   N9:4  SYSTEM_ALARM  "STATE System Alarm" %
%   N15:0  MANUAL_VALVE_NUMBER  "COMMAND HMI The number of the valve under manual control" %
%   B35:2/0  MANUAL_VALVE_OPEN  "COMMAND HMI Open the selected valve" %
%   N15:4/4  MAN_ADS_B_PURIFY_IN  "CONTROL Manually open the bypass valve" %
%   B35:2/1  MANUAL_VALVE_CLOSE  "COMMAND HMI Close the selected valve" %
% Rung: 5 %
SOR BST EQU N10:0 N9:3 NXB EQU N10:0 N9:4 BND BST EQU N15:0 8 XIC B35:2/0 NXB XIC N15:4/5 BND BST XIO B35:2/1 NXB NEQ N15:0 8 BND OTE N15:4/5 EOR
%   N10:0  SYSTEM_STATE  "STATE The current state of the system" %
%   N9:3  SYSTEM_MANUAL  "STATE System Manual" %
%   N9:4  SYSTEM_ALARM  "STATE System Alarm" %
%   N15:0  MANUAL_VALVE_NUMBER  "COMMAND HMI The number of the valve under manual control" %
%   B35:2/0  MANUAL_VALVE_OPEN  "COMMAND HMI Open the selected valve" %
%   N15:4/5  MAN_ADS_B_PURIFY_OUT  "CONTROL Manual Open the regen gas valve" %
%   B35:2/1  MANUAL_VALVE_CLOSE  "COMMAND HMI Close the selected valve" %
% Rung: 6 %
SOR BST EQU N10:0 N9:3 NXB EQU N10:0 N9:4 BND BST EQU N15:0 4 XIC B35:2/0 NXB XIC N15:4/6 BND BST XIO B35:2/1 NXB NEQ N15:0 4 BND OTE N15:4/6 EOR
%   N10:0  SYSTEM_STATE  "STATE The current state of the system" %
%   N9:3  SYSTEM_MANUAL  "STATE System Manual" %
%   N9:4  SYSTEM_ALARM  "STATE System Alarm" %
%   N15:0  MANUAL_VALVE_NUMBER  "COMMAND HMI The number of the valve under manual control" %
%   B35:2/0  MANUAL_VALVE_OPEN  "COMMAND HMI Open the selected valve" %
%   N15:4/6  MAN_ADS_B_REGEN_OUT %
%   B35:2/1  MANUAL_VALVE_CLOSE  "COMMAND HMI Close the selected valve" %
% Rung: 7 %
SOR BST EQU N10:0 N9:3 NXB EQU N10:0 N9:4 BND BST EQU N15:0 9 XIC B35:2/0 NXB XIC N15:4/7 BND BST XIO B35:2/1 NXB NEQ N15:0 9 BND OTE N15:4/7 EOR
%   N10:0  SYSTEM_STATE  "STATE The current state of the system" %
%   N9:3  SYSTEM_MANUAL  "STATE System Manual" %
%   N9:4  SYSTEM_ALARM  "STATE System Alarm" %
%   N15:0  MANUAL_VALVE_NUMBER  "COMMAND HMI The number of the valve under manual control" %
%   B35:2/0  MANUAL_VALVE_OPEN  "COMMAND HMI Open the selected valve" %
%   N15:4/7  MAN_ADS_B_REGEN_IN %
%   B35:2/1  MANUAL_VALVE_CLOSE  "COMMAND HMI Close the selected valve" %

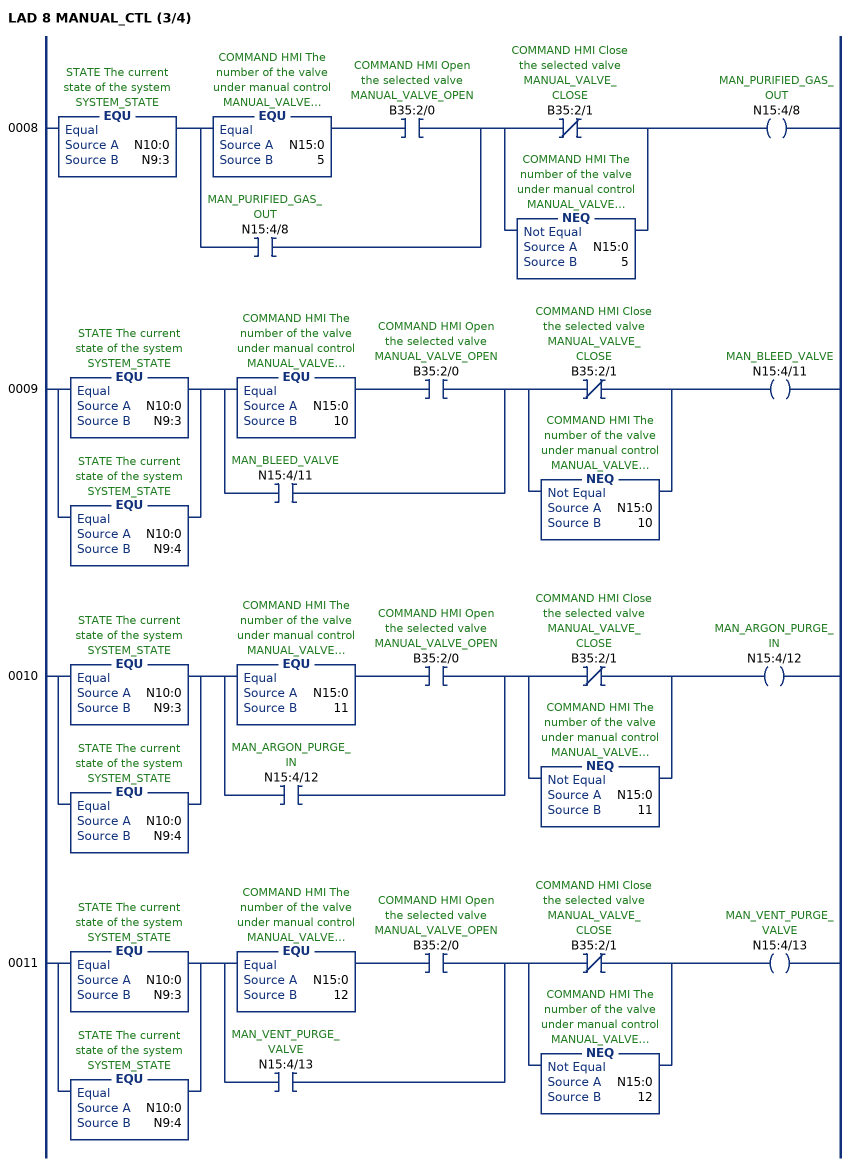
% Rung: 8 %
SOR EQU N10:0 N9:3 BST EQU N15:0 5 XIC B35:2/0 NXB XIC N15:4/8 BND BST XIO B35:2/1 NXB NEQ N15:0 5 BND OTE N15:4/8 EOR
%   N10:0  SYSTEM_STATE  "STATE The current state of the system" %
%   N9:3  SYSTEM_MANUAL  "STATE System Manual" %
%   N15:0  MANUAL_VALVE_NUMBER  "COMMAND HMI The number of the valve under manual control" %
%   B35:2/0  MANUAL_VALVE_OPEN  "COMMAND HMI Open the selected valve" %
%   N15:4/8  MAN_PURIFIED_GAS_OUT %
%   B35:2/1  MANUAL_VALVE_CLOSE  "COMMAND HMI Close the selected valve" %
% Rung: 9 %
SOR BST EQU N10:0 N9:3 NXB EQU N10:0 N9:4 BND BST EQU N15:0 10 XIC B35:2/0 NXB XIC N15:4/11 BND BST XIO B35:2/1 NXB NEQ N15:0 10 BND OTE N15:4/11 EOR
%   N10:0  SYSTEM_STATE  "STATE The current state of the system" %
%   N9:3  SYSTEM_MANUAL  "STATE System Manual" %
%   N9:4  SYSTEM_ALARM  "STATE System Alarm" %
%   N15:0  MANUAL_VALVE_NUMBER  "COMMAND HMI The number of the valve under manual control" %
%   B35:2/0  MANUAL_VALVE_OPEN  "COMMAND HMI Open the selected valve" %
%   N15:4/11  MAN_BLEED_VALVE %
%   B35:2/1  MANUAL_VALVE_CLOSE  "COMMAND HMI Close the selected valve" %
% Rung: 10 %
SOR BST EQU N10:0 N9:3 NXB EQU N10:0 N9:4 BND BST EQU N15:0 11 XIC B35:2/0 NXB XIC N15:4/12 BND BST XIO B35:2/1 NXB NEQ N15:0 11 BND OTE N15:4/12 EOR
%   N10:0  SYSTEM_STATE  "STATE The current state of the system" %
%   N9:3  SYSTEM_MANUAL  "STATE System Manual" %
%   N9:4  SYSTEM_ALARM  "STATE System Alarm" %
%   N15:0  MANUAL_VALVE_NUMBER  "COMMAND HMI The number of the valve under manual control" %
%   B35:2/0  MANUAL_VALVE_OPEN  "COMMAND HMI Open the selected valve" %
%   N15:4/12  MAN_ARGON_PURGE_IN %
%   B35:2/1  MANUAL_VALVE_CLOSE  "COMMAND HMI Close the selected valve" %
% Rung: 11 %
SOR BST EQU N10:0 N9:3 NXB EQU N10:0 N9:4 BND BST EQU N15:0 12 XIC B35:2/0 NXB XIC N15:4/13 BND BST XIO B35:2/1 NXB NEQ N15:0 12 BND OTE N15:4/13 EOR
%   N10:0  SYSTEM_STATE  "STATE The current state of the system" %
%   N9:3  SYSTEM_MANUAL  "STATE System Manual" %
%   N9:4  SYSTEM_ALARM  "STATE System Alarm" %
%   N15:0  MANUAL_VALVE_NUMBER  "COMMAND HMI The number of the valve under manual control" %
%   B35:2/0  MANUAL_VALVE_OPEN  "COMMAND HMI Open the selected valve" %
%   N15:4/13  MAN_VENT_PURGE_VALVE %
%   B35:2/1  MANUAL_VALVE_CLOSE  "COMMAND HMI Close the selected valve" %

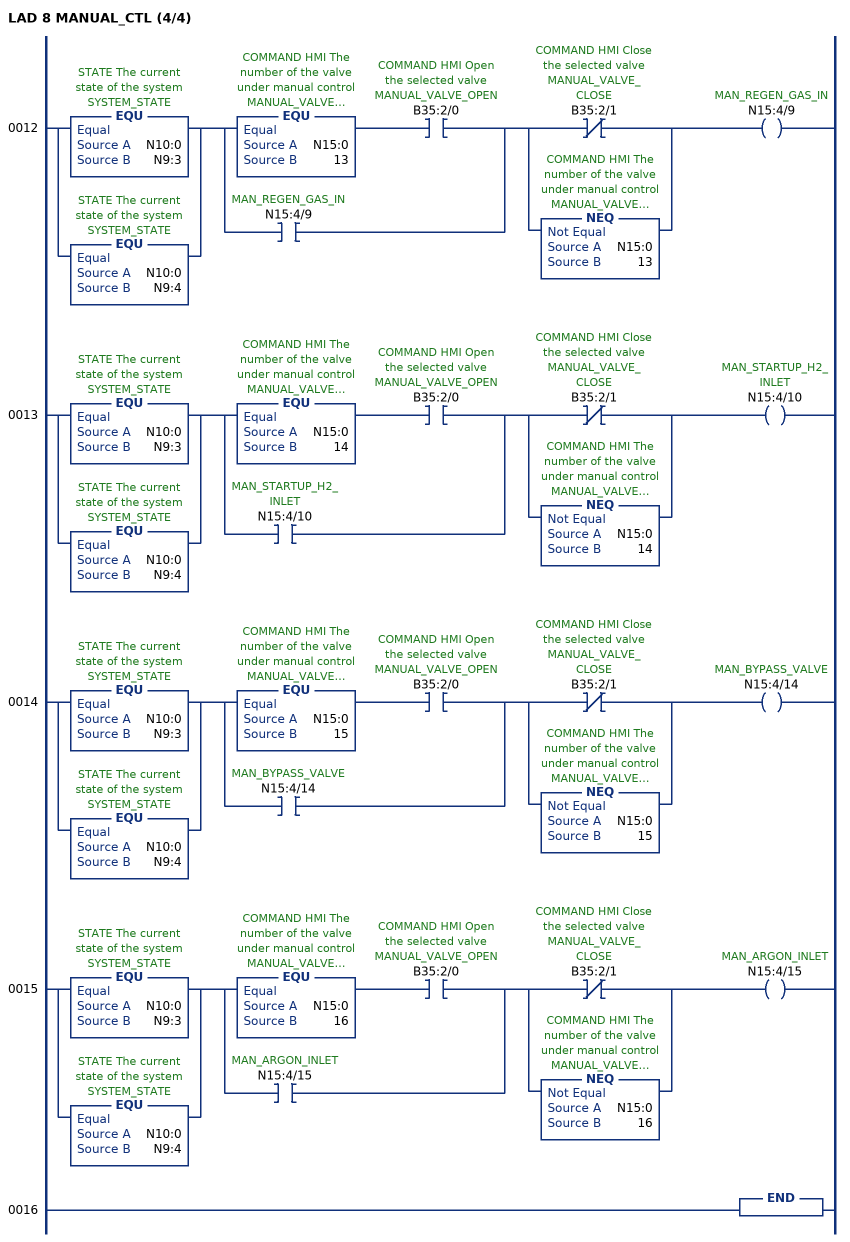
% Rung: 12 %
SOR BST EQU N10:0 N9:3 NXB EQU N10:0 N9:4 BND BST EQU N15:0 13 XIC B35:2/0 NXB XIC N15:4/9 BND BST XIO B35:2/1 NXB NEQ N15:0 13 BND OTE N15:4/9 EOR
%   N10:0  SYSTEM_STATE  "STATE The current state of the system" %
%   N9:3  SYSTEM_MANUAL  "STATE System Manual" %
%   N9:4  SYSTEM_ALARM  "STATE System Alarm" %
%   N15:0  MANUAL_VALVE_NUMBER  "COMMAND HMI The number of the valve under manual control" %
%   B35:2/0  MANUAL_VALVE_OPEN  "COMMAND HMI Open the selected valve" %
%   N15:4/9  MAN_REGEN_GAS_IN %
%   B35:2/1  MANUAL_VALVE_CLOSE  "COMMAND HMI Close the selected valve" %
% Rung: 13 %
SOR BST EQU N10:0 N9:3 NXB EQU N10:0 N9:4 BND BST EQU N15:0 14 XIC B35:2/0 NXB XIC N15:4/10 BND BST XIO B35:2/1 NXB NEQ N15:0 14 BND OTE N15:4/10 EOR
%   N10:0  SYSTEM_STATE  "STATE The current state of the system" %
%   N9:3  SYSTEM_MANUAL  "STATE System Manual" %
%   N9:4  SYSTEM_ALARM  "STATE System Alarm" %
%   N15:0  MANUAL_VALVE_NUMBER  "COMMAND HMI The number of the valve under manual control" %
%   B35:2/0  MANUAL_VALVE_OPEN  "COMMAND HMI Open the selected valve" %
%   N15:4/10  MAN_STARTUP_H2_INLET %
%   B35:2/1  MANUAL_VALVE_CLOSE  "COMMAND HMI Close the selected valve" %
% Rung: 14 %
SOR BST EQU N10:0 N9:3 NXB EQU N10:0 N9:4 BND BST EQU N15:0 15 XIC B35:2/0 NXB XIC N15:4/14 BND BST XIO B35:2/1 NXB NEQ N15:0 15 BND OTE N15:4/14 EOR
%   N10:0  SYSTEM_STATE  "STATE The current state of the system" %
%   N9:3  SYSTEM_MANUAL  "STATE System Manual" %
%   N9:4  SYSTEM_ALARM  "STATE System Alarm" %
%   N15:0  MANUAL_VALVE_NUMBER  "COMMAND HMI The number of the valve under manual control" %
%   B35:2/0  MANUAL_VALVE_OPEN  "COMMAND HMI Open the selected valve" %
%   N15:4/14  MAN_BYPASS_VALVE %
%   B35:2/1  MANUAL_VALVE_CLOSE  "COMMAND HMI Close the selected valve" %
% Rung: 15 %
SOR BST EQU N10:0 N9:3 NXB EQU N10:0 N9:4 BND BST EQU N15:0 16 XIC B35:2/0 NXB XIC N15:4/15 BND BST XIO B35:2/1 NXB NEQ N15:0 16 BND OTE N15:4/15 EOR
%   N10:0  SYSTEM_STATE  "STATE The current state of the system" %
%   N9:3  SYSTEM_MANUAL  "STATE System Manual" %
%   N9:4  SYSTEM_ALARM  "STATE System Alarm" %
%   N15:0  MANUAL_VALVE_NUMBER  "COMMAND HMI The number of the valve under manual control" %
%   B35:2/0  MANUAL_VALVE_OPEN  "COMMAND HMI Open the selected valve" %
%   N15:4/15  MAN_ARGON_INLET %
%   B35:2/1  MANUAL_VALVE_CLOSE  "COMMAND HMI Close the selected valve" %
% Rung: 16 %
SOR END EOR

LADDER 9 "STARTUP"
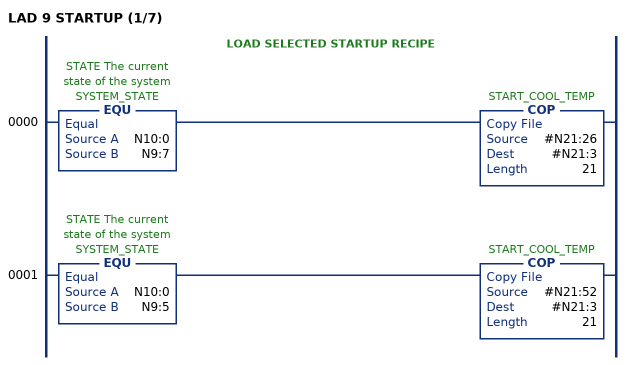
% Rung: 0 %
% TITLE: LOAD SELECTED STARTUP RECIPE %
SOR EQU N10:0 N9:7 COP #N21:26 #N21:3 21 EOR
%   N10:0  SYSTEM_STATE  "STATE The current state of the system" %
%   N9:7  SYSTEM_COLD_START %
%   N21:26  COLD_COOL_TEMP %
%   N21:3  START_COOL_TEMP %
% Rung: 1 %
SOR EQU N10:0 N9:5 COP #N21:52 #N21:3 21 EOR
%   N10:0  SYSTEM_STATE  "STATE The current state of the system" %
%   N9:5  SYSTEM_QUICK_START %
%   N21:52  QUICK_COOL_TEMP %
%   N21:3  START_COOL_TEMP %

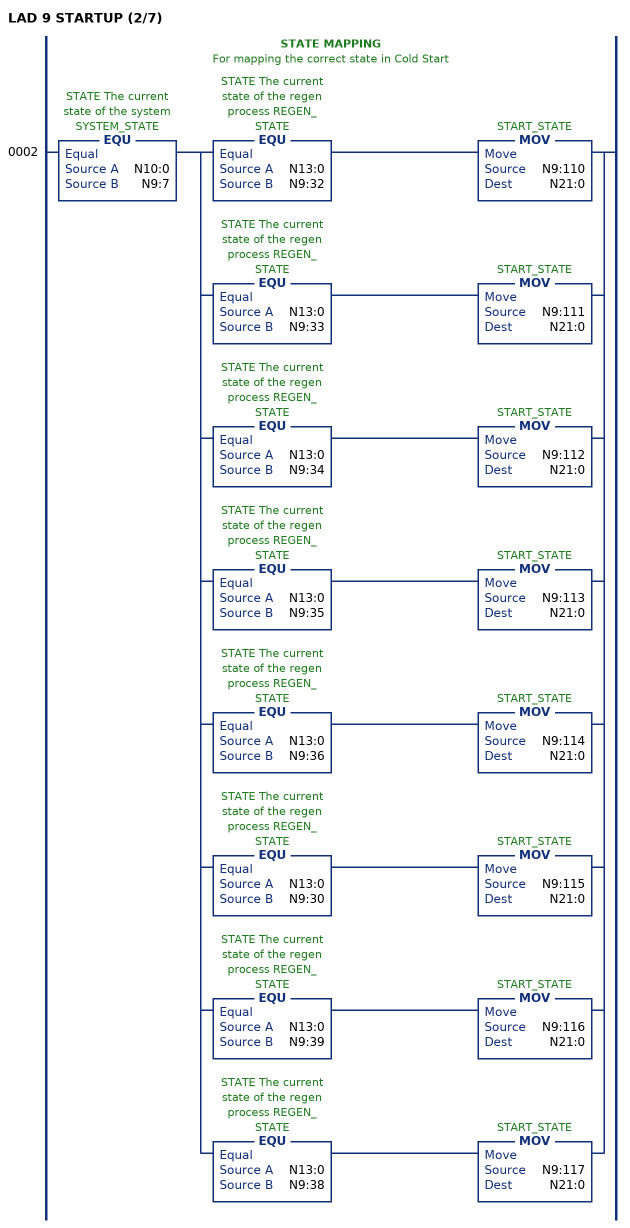
% Rung: 2 %
% TITLE: STATE MAPPING %
% For mapping the correct state in Cold Start %
SOR EQU N10:0 N9:7 BST EQU N13:0 N9:32 MOV N9:110 N21:0 NXB EQU N13:0 N9:33 MOV N9:111 N21:0 NXB EQU N13:0 N9:34 MOV N9:112 N21:0 NXB EQU N13:0 N9:35 MOV N9:113 N21:0 NXB EQU N13:0 N9:36 MOV N9:114 N21:0 NXB EQU N13:0 N9:30 MOV N9:115 N21:0 NXB EQU N13:0 N9:39 MOV N9:116 N21:0 NXB EQU N13:0 N9:38 MOV N9:117 N21:0 BND EOR
%   N10:0  SYSTEM_STATE  "STATE The current state of the system" %
%   N9:7  SYSTEM_COLD_START %
%   N13:0  REGEN_STATE  "STATE The current state of the regen process" %
%   N9:32  REGEN_VENT  "STATE Regen Vent" %
%   N9:110  START_REG_VENT %
%   N21:0  START_STATE %
%   N9:33  REGEN_HEAT_BED  "STATE Regen Heat wall" %
%   N9:111  START_REG_HEAT %
%   N9:34  REGEN_RUN  "STATE Regen Running" %
%   N9:112  START_REG_RUN %
%   N9:35  REGEN_COOL_WALL  "STATE Regen Cool wall" %
%   N9:113  START_REG_COOL %
%   N9:36  REGEN_COOL  "STATE Regen Cool" %
%   N9:114  START_REG_TIMED_COOL %
%   N9:30  REGEN_STANDBY  "STATE Regen Standby" %
%   N9:115  START_REG_STANDBY %
%   N9:39  REGEN_BACKFILL %
%   N9:116  START_REG_BACKFILL %
%   N9:38  REGEN_DONE %
%   N9:117  START_REG_DONE %

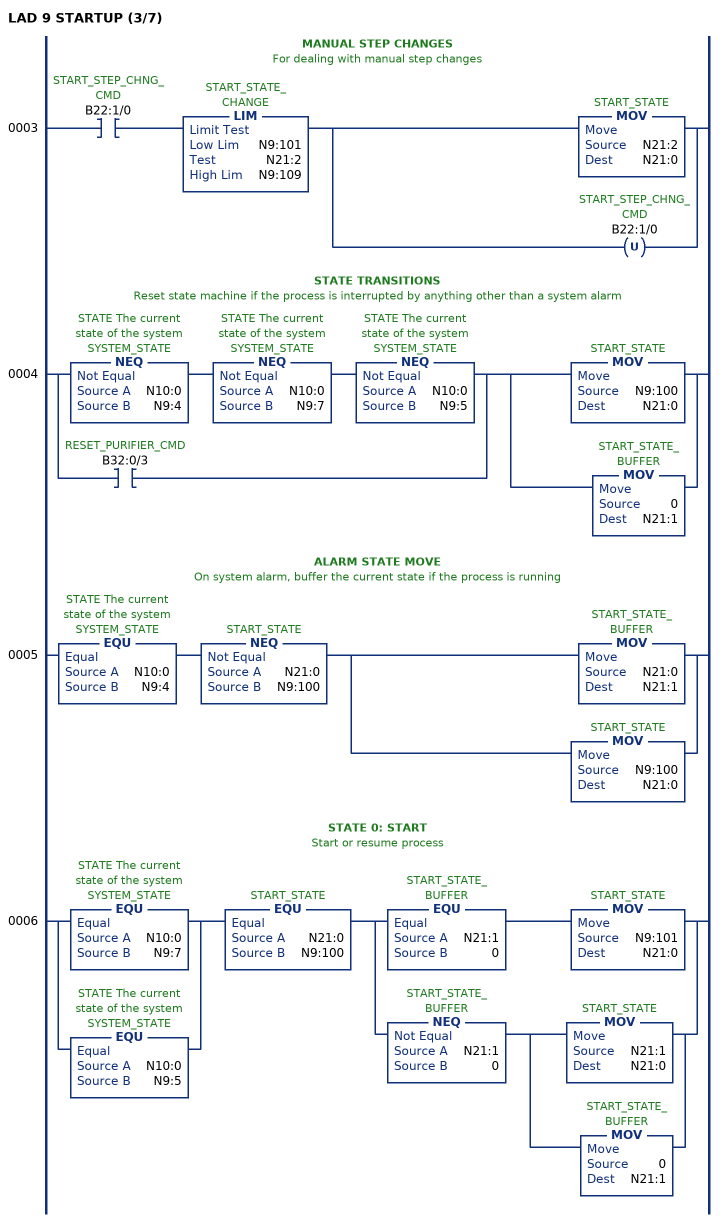
% Rung: 3 %
% TITLE: MANUAL STEP CHANGES %
% For dealing with manual step changes %
SOR XIC B22:1/0 LIM N9:101 N21:2 N9:109 BST MOV N21:2 N21:0 NXB OTU B22:1/0 BND EOR
%   B22:1/0  START_STEP_CHNG_CMD %
%   N9:101  START_COOL %
%   N21:2  START_STATE_CHANGE %
%   N9:109  START_BACKFILL_2 %
%   N21:0  START_STATE %
% Rung: 4 %
% TITLE: STATE TRANSITIONS %
% Reset state machine if the process is interrupted by anything other than a system alarm %
SOR BST NEQ N10:0 N9:4 NEQ N10:0 N9:7 NEQ N10:0 N9:5 NXB XIC B32:0/3 BND BST MOV N9:100 N21:0 NXB MOV 0 N21:1 BND EOR
%   N10:0  SYSTEM_STATE  "STATE The current state of the system" %
%   N9:4  SYSTEM_ALARM  "STATE System Alarm" %
%   N9:7  SYSTEM_COLD_START %
%   N9:5  SYSTEM_QUICK_START %
%   B32:0/3  RESET_PURIFIER_CMD %
%   N9:100  START_IDLE %
%   N21:0  START_STATE %
%   N21:1  START_STATE_BUFFER %
% Rung: 5 %
% TITLE: ALARM STATE MOVE %
% On system alarm, buffer the current state if the process is running %
SOR EQU N10:0 N9:4 NEQ N21:0 N9:100 BST MOV N21:0 N21:1 NXB MOV N9:100 N21:0 BND EOR
%   N10:0  SYSTEM_STATE  "STATE The current state of the system" %
%   N9:4  SYSTEM_ALARM  "STATE System Alarm" %
%   N21:0  START_STATE %
%   N9:100  START_IDLE %
%   N21:1  START_STATE_BUFFER %
% Rung: 6 %
% TITLE: STATE 0: START %
% Start or resume process %
SOR BST EQU N10:0 N9:7 NXB EQU N10:0 N9:5 BND EQU N21:0 N9:100 BST EQU N21:1 0 MOV N9:101 N21:0 NXB NEQ N21:1 0 BST MOV N21:1 N21:0 NXB MOV 0 N21:1 BND BND EOR
%   N10:0  SYSTEM_STATE  "STATE The current state of the system" %
%   N9:7  SYSTEM_COLD_START %
%   N9:5  SYSTEM_QUICK_START %
%   N21:0  START_STATE %
%   N9:100  START_IDLE %
%   N21:1  START_STATE_BUFFER %
%   N9:101  START_COOL %

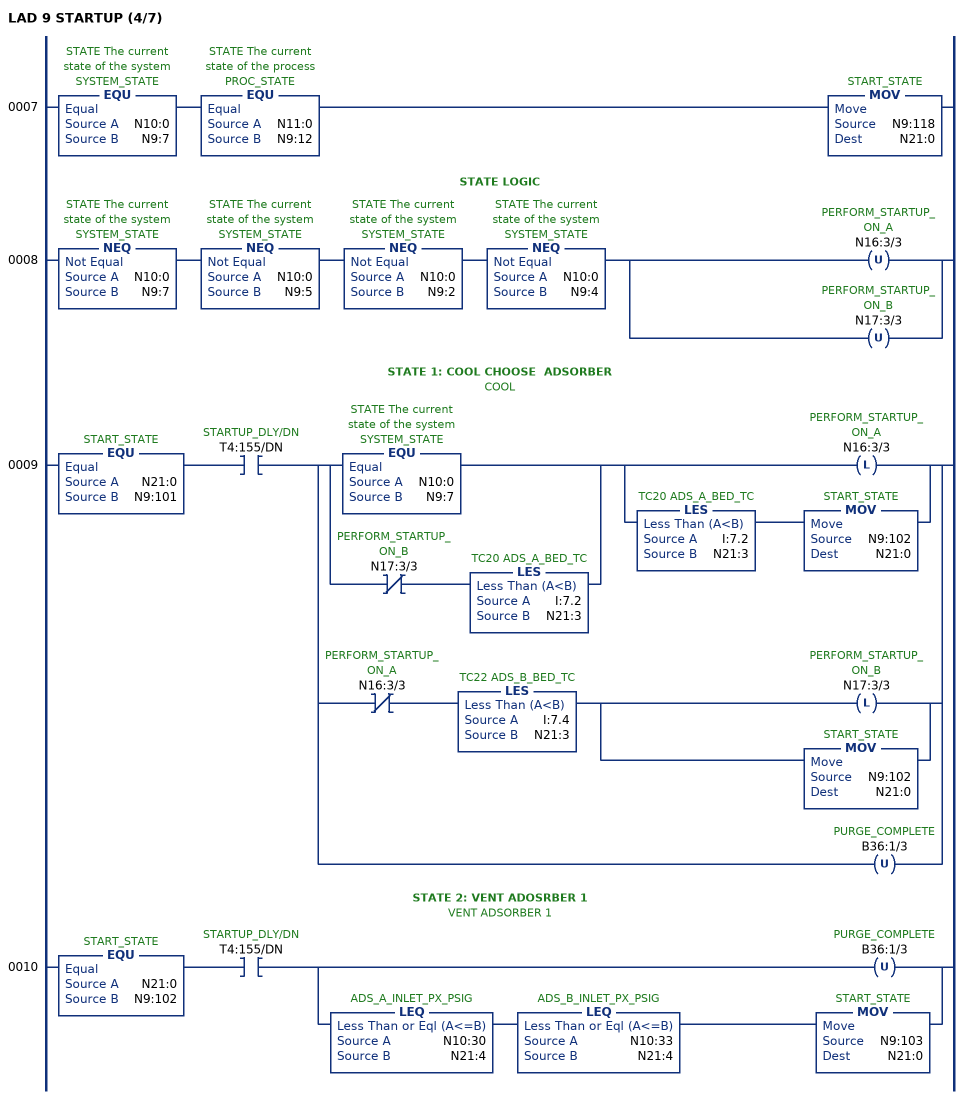
% Rung: 7 %
SOR EQU N10:0 N9:7 EQU N11:0 N9:12 MOV N9:118 N21:0 EOR
%   N10:0  SYSTEM_STATE  "STATE The current state of the system" %
%   N9:7  SYSTEM_COLD_START %
%   N11:0  PROC_STATE  "STATE The current state of the process" %
%   N9:12  PROC_PFY_B_REG_A  "STATE Process Purify B" %
%   N9:118  START_DONE %
%   N21:0  START_STATE %
% Rung: 8 %
% TITLE: STATE LOGIC %
SOR NEQ N10:0 N9:7 NEQ N10:0 N9:5 NEQ N10:0 N9:2 NEQ N10:0 N9:4 BST OTU N16:3/3 NXB OTU N17:3/3 BND EOR
%   N10:0  SYSTEM_STATE  "STATE The current state of the system" %
%   N9:7  SYSTEM_COLD_START %
%   N9:5  SYSTEM_QUICK_START %
%   N9:2  SYSTEM_PROCESS  "STATE System Process" %
%   N9:4  SYSTEM_ALARM  "STATE System Alarm" %
%   N16:3/3  PERFORM_STARTUP_ON_A %
%   N17:3/3  PERFORM_STARTUP_ON_B %
% Rung: 9 %
% TITLE: STATE 1: COOL CHOOSE  ADSORBER %
% COOL %
SOR EQU N21:0 N9:101 XIC T4:155/DN BST BST EQU N10:0 N9:7 NXB XIO N17:3/3 LES I:7.2 N21:3 BND BST OTL N16:3/3 NXB LES I:7.2 N21:3 MOV N9:102 N21:0 BND NXB XIO N16:3/3 LES I:7.4 N21:3 BST OTL N17:3/3 NXB MOV N9:102 N21:0 BND NXB OTU B36:1/3 BND EOR
%   N21:0  START_STATE %
%   N9:101  START_COOL %
%   T4:155  STARTUP_DLY %
%   N10:0  SYSTEM_STATE  "STATE The current state of the system" %
%   N9:7  SYSTEM_COLD_START %
%   N17:3/3  PERFORM_STARTUP_ON_B %
%   I:7.2  ADS_A_BED_TC  "TC20" %
%   N21:3  START_COOL_TEMP %
%   N16:3/3  PERFORM_STARTUP_ON_A %
%   N9:102  START_VENT_ADS_1 %
%   I:7.4  ADS_B_BED_TC  "TC22" %
%   B36:1/3  PURGE_COMPLETE %
% Rung: 10 %
% TITLE: STATE 2: VENT ADOSRBER 1 %
% VENT ADSORBER 1 %
SOR EQU N21:0 N9:102 XIC T4:155/DN BST OTU B36:1/3 NXB LEQ N10:30 N21:4 LEQ N10:33 N21:4 MOV N9:103 N21:0 BND EOR
%   N21:0  START_STATE %
%   N9:102  START_VENT_ADS_1 %
%   T4:155  STARTUP_DLY %
%   B36:1/3  PURGE_COMPLETE %
%   N10:30  ADS_A_INLET_PX_PSIG %
%   N21:4  START_VENT_ADS_1_PRS %
%   N10:33  ADS_B_INLET_PX_PSIG %
%   N9:103  START_VENT_GET_1 %

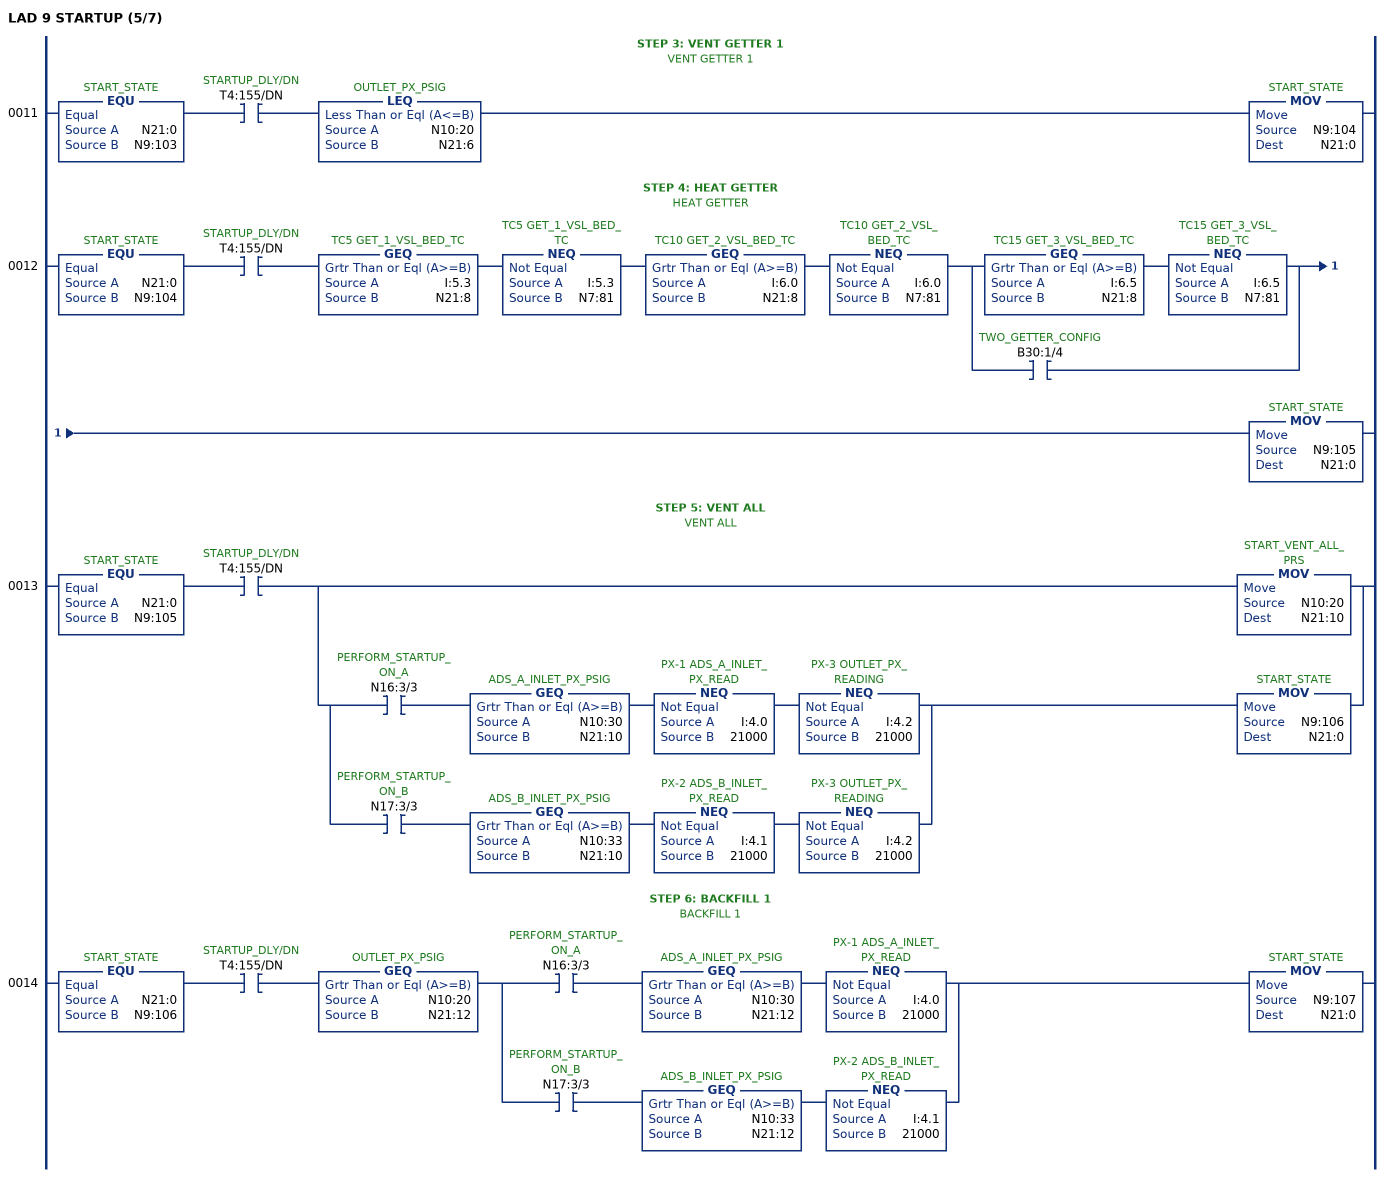
% Rung: 11 %
% TITLE: STEP 3: VENT GETTER 1 %
% VENT GETTER 1 %
SOR EQU N21:0 N9:103 XIC T4:155/DN LEQ N10:20 N21:6 MOV N9:104 N21:0 EOR
%   N21:0  START_STATE %
%   N9:103  START_VENT_GET_1 %
%   T4:155  STARTUP_DLY %
%   N10:20  OUTLET_PX_PSIG %
%   N21:6  START_VENT_GET_1_PRS %
%   N9:104  START_HEAT %
% Rung: 12 %
% TITLE: STEP 4: HEAT GETTER %
% HEAT GETTER %
SOR EQU N21:0 N9:104 XIC T4:155/DN GEQ I:5.3 N21:8 NEQ I:5.3 N7:81 GEQ I:6.0 N21:8 NEQ I:6.0 N7:81 BST GEQ I:6.5 N21:8 NEQ I:6.5 N7:81 NXB XIC B30:1/4 BND MOV N9:105 N21:0 EOR
%   N21:0  START_STATE %
%   N9:104  START_HEAT %
%   T4:155  STARTUP_DLY %
%   I:5.3  GET_1_VSL_BED_TC  "TC5" %
%   N21:8  START_HEAT_TEMP %
%   N7:81  TC_OPEN_SP  "CONFIG The value read by an open TC input" %
%   I:6.0  GET_2_VSL_BED_TC  "TC10" %
%   I:6.5  GET_3_VSL_BED_TC  "TC15" %
%   B30:1/4  TWO_GETTER_CONFIG %
%   N9:105  START_VENT_ALL %
% Rung: 13 %
% TITLE: STEP 5: VENT ALL %
% VENT ALL %
SOR EQU N21:0 N9:105 XIC T4:155/DN BST MOV N10:20 N21:10 NXB BST XIC N16:3/3 GEQ N10:30 N21:10 NEQ I:4.0 21000 NEQ I:4.2 21000 NXB XIC N17:3/3 GEQ N10:33 N21:10 NEQ I:4.1 21000 NEQ I:4.2 21000 BND MOV N9:106 N21:0 BND EOR
%   N21:0  START_STATE %
%   N9:105  START_VENT_ALL %
%   T4:155  STARTUP_DLY %
%   N10:20  OUTLET_PX_PSIG %
%   N21:10  START_VENT_ALL_PRS %
%   N16:3/3  PERFORM_STARTUP_ON_A %
%   N10:30  ADS_A_INLET_PX_PSIG %
%   I:4.0  ADS_A_INLET_PX_READ  "PX-1" %
%   I:4.2  OUTLET_PX_READING  "PX-3" %
%   N17:3/3  PERFORM_STARTUP_ON_B %
%   N10:33  ADS_B_INLET_PX_PSIG %
%   I:4.1  ADS_B_INLET_PX_READ  "PX-2" %
%   N9:106  START_BACKFILL_1 %
% Rung: 14 %
% TITLE: STEP 6: BACKFILL 1 %
% BACKFILL 1 %
SOR EQU N21:0 N9:106 XIC T4:155/DN GEQ N10:20 N21:12 BST XIC N16:3/3 GEQ N10:30 N21:12 NEQ I:4.0 21000 NXB XIC N17:3/3 GEQ N10:33 N21:12 NEQ I:4.1 21000 BND MOV N9:107 N21:0 EOR
%   N21:0  START_STATE %
%   N9:106  START_BACKFILL_1 %
%   T4:155  STARTUP_DLY %
%   N10:20  OUTLET_PX_PSIG %
%   N21:12  START_BKFIL_1_PRS %
%   N16:3/3  PERFORM_STARTUP_ON_A %
%   N10:30  ADS_A_INLET_PX_PSIG %
%   I:4.0  ADS_A_INLET_PX_READ  "PX-1" %
%   N17:3/3  PERFORM_STARTUP_ON_B %
%   N10:33  ADS_B_INLET_PX_PSIG %
%   I:4.1  ADS_B_INLET_PX_READ  "PX-2" %
%   N9:107  START_VENT_ADS_2 %

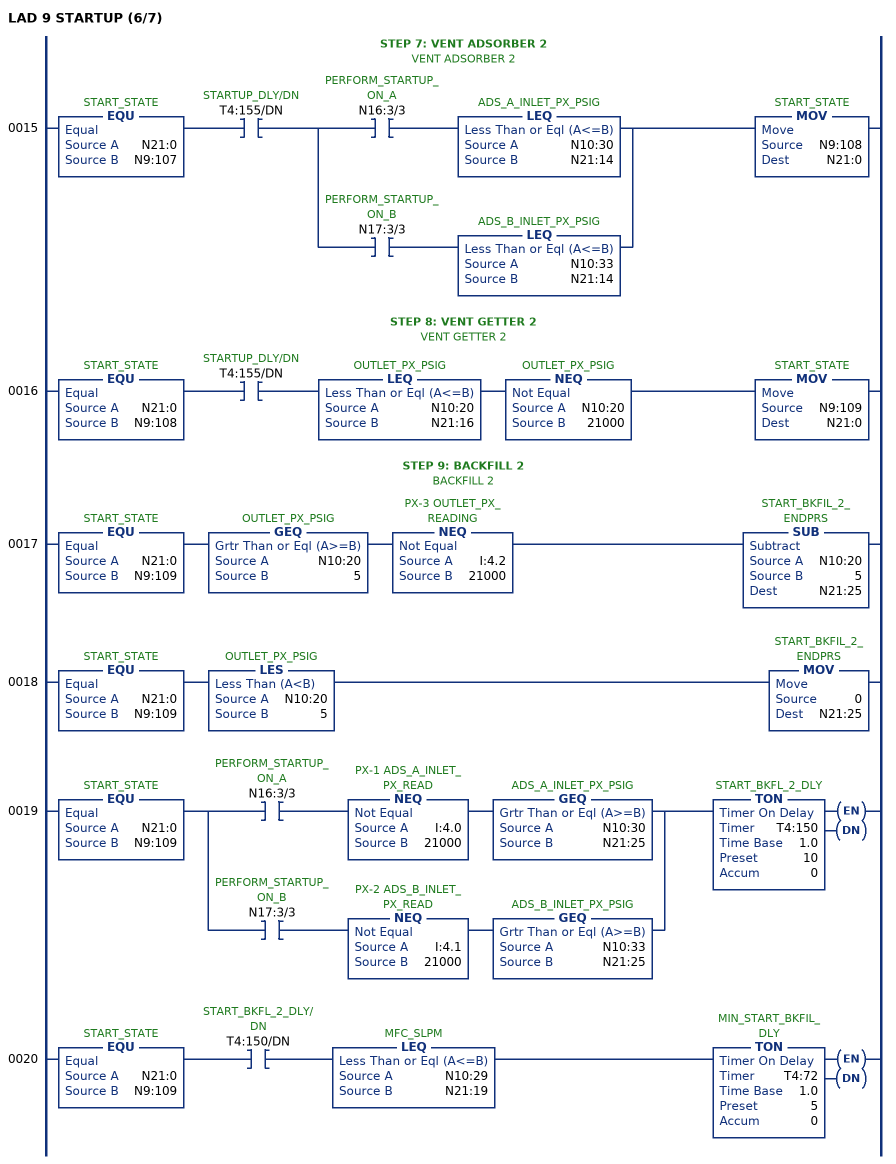
% Rung: 15 %
% TITLE: STEP 7: VENT ADSORBER 2 %
% VENT ADSORBER 2 %
SOR EQU N21:0 N9:107 XIC T4:155/DN BST XIC N16:3/3 LEQ N10:30 N21:14 NXB XIC N17:3/3 LEQ N10:33 N21:14 BND MOV N9:108 N21:0 EOR
%   N21:0  START_STATE %
%   N9:107  START_VENT_ADS_2 %
%   T4:155  STARTUP_DLY %
%   N16:3/3  PERFORM_STARTUP_ON_A %
%   N10:30  ADS_A_INLET_PX_PSIG %
%   N21:14  START_VENT_ADS_2_PRS %
%   N17:3/3  PERFORM_STARTUP_ON_B %
%   N10:33  ADS_B_INLET_PX_PSIG %
%   N9:108  START_VENT_GET_2 %
% Rung: 16 %
% TITLE: STEP 8: VENT GETTER 2 %
% VENT GETTER 2 %
SOR EQU N21:0 N9:108 XIC T4:155/DN LEQ N10:20 N21:16 NEQ N10:20 21000 MOV N9:109 N21:0 EOR
%   N21:0  START_STATE %
%   N9:108  START_VENT_GET_2 %
%   T4:155  STARTUP_DLY %
%   N10:20  OUTLET_PX_PSIG %
%   N21:16  START_VENT_GET_2_PRS %
%   N9:109  START_BACKFILL_2 %
% Rung: 17 %
% TITLE: STEP 9: BACKFILL 2 %
% BACKFILL 2 %
SOR EQU N21:0 N9:109 GEQ N10:20 5 NEQ I:4.2 21000 SUB N10:20 5 N21:25 EOR
%   N21:0  START_STATE %
%   N9:109  START_BACKFILL_2 %
%   N10:20  OUTLET_PX_PSIG %
%   I:4.2  OUTLET_PX_READING  "PX-3" %
%   N21:25  START_BKFIL_2_ENDPRS %
% Rung: 18 %
SOR EQU N21:0 N9:109 LES N10:20 5 MOV 0 N21:25 EOR
%   N21:0  START_STATE %
%   N9:109  START_BACKFILL_2 %
%   N10:20  OUTLET_PX_PSIG %
%   N21:25  START_BKFIL_2_ENDPRS %
% Rung: 19 %
SOR EQU N21:0 N9:109 BST XIC N16:3/3 NEQ I:4.0 21000 GEQ N10:30 N21:25 NXB XIC N17:3/3 NEQ I:4.1 21000 GEQ N10:33 N21:25 BND TON T4:150 1.0 10 0 EOR
%   N21:0  START_STATE %
%   N9:109  START_BACKFILL_2 %
%   N16:3/3  PERFORM_STARTUP_ON_A %
%   I:4.0  ADS_A_INLET_PX_READ  "PX-1" %
%   N10:30  ADS_A_INLET_PX_PSIG %
%   N21:25  START_BKFIL_2_ENDPRS %
%   N17:3/3  PERFORM_STARTUP_ON_B %
%   I:4.1  ADS_B_INLET_PX_READ  "PX-2" %
%   N10:33  ADS_B_INLET_PX_PSIG %
%   T4:150  START_BKFL_2_DLY %
% Rung: 20 %
SOR EQU N21:0 N9:109 XIC T4:150/DN LEQ N10:29 N21:19 TON T4:72 1.0 5 0 EOR
%   N21:0  START_STATE %
%   N9:109  START_BACKFILL_2 %
%   T4:150  START_BKFL_2_DLY %
%   N10:29  MFC_SLPM %
%   N21:19  START_BKFIL_2_ENDFLW %
%   T4:72  MIN_START_BKFIL_DLY %

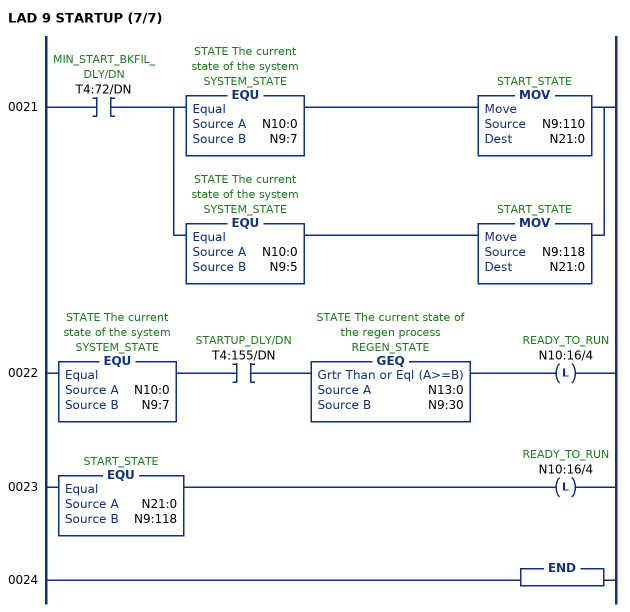
% Rung: 21 %
SOR XIC T4:72/DN BST EQU N10:0 N9:7 MOV N9:110 N21:0 NXB EQU N10:0 N9:5 MOV N9:118 N21:0 BND EOR
%   T4:72  MIN_START_BKFIL_DLY %
%   N10:0  SYSTEM_STATE  "STATE The current state of the system" %
%   N9:7  SYSTEM_COLD_START %
%   N9:110  START_REG_VENT %
%   N21:0  START_STATE %
%   N9:5  SYSTEM_QUICK_START %
%   N9:118  START_DONE %
% Rung: 22 %
SOR EQU N10:0 N9:7 XIC T4:155/DN GEQ N13:0 N9:30 OTL N10:16/4 EOR
%   N10:0  SYSTEM_STATE  "STATE The current state of the system" %
%   N9:7  SYSTEM_COLD_START %
%   T4:155  STARTUP_DLY %
%   N13:0  REGEN_STATE  "STATE The current state of the regen process" %
%   N9:30  REGEN_STANDBY  "STATE Regen Standby" %
%   N10:16/4  READY_TO_RUN %
% Rung: 23 %
SOR EQU N21:0 N9:118 OTL N10:16/4 EOR
%   N21:0  START_STATE %
%   N9:118  START_DONE %
%   N10:16/4  READY_TO_RUN %
% Rung: 24 %
SOR END EOR

LADDER 10 "PURIFY"    % Operates the purify control %
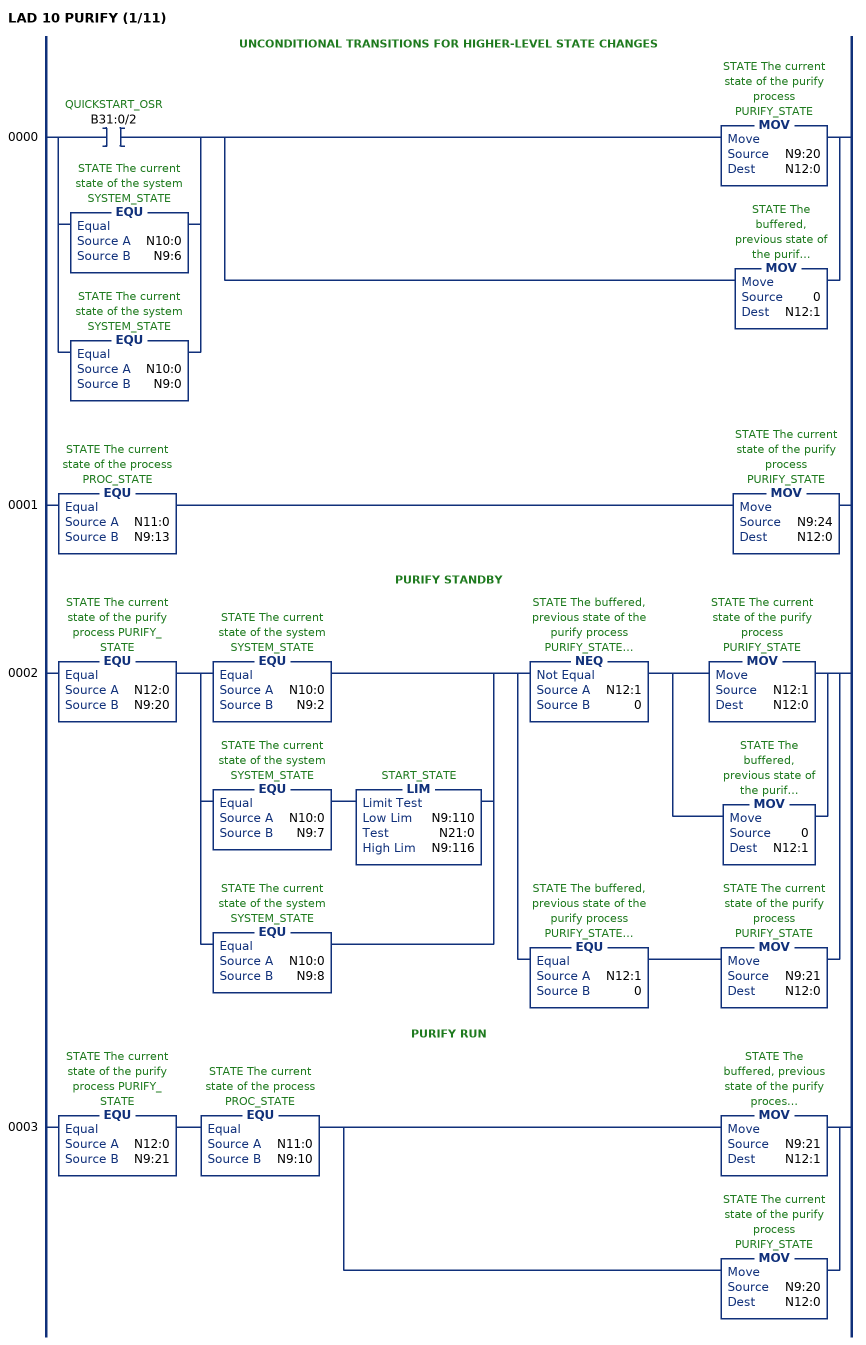
% Rung: 0 %
% TITLE: UNCONDITIONAL TRANSITIONS FOR HIGHER-LEVEL STATE CHANGES %
SOR BST XIC B31:0/2 NXB EQU N10:0 N9:6 NXB EQU N10:0 N9:0 BND BST MOV N9:20 N12:0 NXB MOV 0 N12:1 BND EOR
%   B31:0/2  QUICKSTART_OSR %
%   N10:0  SYSTEM_STATE  "STATE The current state of the system" %
%   N9:6  SYSTEM_PURGE %
%   N9:0  SYSTEM_OFFLINE %
%   N9:20  PURIFY_STANDBY  "STATE Purify Standby" %
%   N12:0  PURIFY_STATE  "STATE The current state of the purify process" %
%   N12:1  PURIFY_STATE_BUFFER  "STATE The buffered, previous state of the purify process" %
% Rung: 1 %
SOR EQU N11:0 N9:13 MOV N9:24 N12:0 EOR
%   N11:0  PROC_STATE  "STATE The current state of the process" %
%   N9:13  PROC_OVERLAP  "STATE Process Purify Overlap" %
%   N9:24  PURIFY_OVERLAP  "STATE Puriify Overlap" %
%   N12:0  PURIFY_STATE  "STATE The current state of the purify process" %
% Rung: 2 %
% TITLE: PURIFY STANDBY %
SOR EQU N12:0 N9:20 BST EQU N10:0 N9:2 NXB EQU N10:0 N9:7 LIM N9:110 N21:0 N9:116 NXB EQU N10:0 N9:8 BND BST NEQ N12:1 0 BST MOV N12:1 N12:0 NXB MOV 0 N12:1 BND NXB EQU N12:1 0 MOV N9:21 N12:0 BND EOR
%   N12:0  PURIFY_STATE  "STATE The current state of the purify process" %
%   N9:20  PURIFY_STANDBY  "STATE Purify Standby" %
%   N10:0  SYSTEM_STATE  "STATE The current state of the system" %
%   N9:2  SYSTEM_PROCESS  "STATE System Process" %
%   N9:7  SYSTEM_COLD_START %
%   N9:110  START_REG_VENT %
%   N21:0  START_STATE %
%   N9:116  START_REG_BACKFILL %
%   N9:8  SYSTEM_SUPPLEMENTAL %
%   N12:1  PURIFY_STATE_BUFFER  "STATE The buffered, previous state of the purify process" %
%   N9:21  PURIFY_RUN  "STATE Purify running" %
% Rung: 3 %
% TITLE: PURIFY RUN %
SOR EQU N12:0 N9:21 EQU N11:0 N9:10 BST MOV N9:21 N12:1 NXB MOV N9:20 N12:0 BND EOR
%   N12:0  PURIFY_STATE  "STATE The current state of the purify process" %
%   N9:21  PURIFY_RUN  "STATE Purify running" %
%   N11:0  PROC_STATE  "STATE The current state of the process" %
%   N9:10  PROC_STANDBY  "STATE Process Standby" %
%   N12:1  PURIFY_STATE_BUFFER  "STATE The buffered, previous state of the purify process" %
%   N9:20  PURIFY_STANDBY  "STATE Purify Standby" %

